C01815=1196.724,348.587,-75.076,-176.172,7.976,148.435
C01816=1196.728,348.340,-75.043,-176.174,7.973,148.435
C01817=1196.731,348.092,-75.011,-176.176,7.970,148.435
C01818=1196.736,347.844,-74.978,-176.177,7.966,148.434
C01819=1196.740,347.596,-74.944,-176.180,7.963,148.434
C01820=1196.745,347.348,-74.912,-176.182,7.960,148.434
C01821=1196.749,347.101,-74.879,-176.184,7.957,148.434
C01822=1196.753,346.853,-74.847,-176.186,7.954,148.433
C01823=1196.757,346.605,-74.814,-176.188,7.951,148.433
C01824=1196.761,346.357,-74.781,-176.190,7.947,148.433
C01825=1196.765,346.109,-74.749,-176.192,7.945,148.433
C01826=1196.769,345.862,-74.716,-176.194,7.941,148.433
C01827=1196.773,345.613,-74.684,-176.196,7.938,148.432
C01828=1196.778,345.366,-74.651,-176.199,7.935,148.432
C01829=1196.782,345.118,-74.619,-176.201,7.931,148.432
C01830=1196.786,344.870,-74.586,-176.202,7.929,148.432
C01831=1196.790,344.622,-74.553,-176.205,7.926,148.431
C01832=1196.794,344.375,-74.521,-176.207,7.922,148.431
C01833=1196.798,344.126,-74.488,-176.209,7.919,148.431
C01834=1196.802,343.879,-74.455,-176.211,7.916,148.431
C01835=1196.807,343.631,-74.424,-176.213,7.913,148.431
C01836=1196.811,343.383,-74.391,-176.216,7.910,148.431
C01837=1196.815,343.135,-74.358,-176.218,7.907,148.430
C01838=1196.819,342.888,-74.326,-176.220,7.904,148.430
C01839=1196.823,342.639,-74.293,-176.222,7.901,148.430
C01840=1196.827,342.391,-74.261,-176.224,7.898,148.430
C01841=1196.831,342.144,-74.228,-176.226,7.894,148.430
C01842=1196.836,341.896,-74.196,-176.228,7.892,148.429
C01843=1196.839,341.648,-74.163,-176.230,7.888,148.429
C01844=1196.844,341.400,-74.131,-176.233,7.885,148.429
C01845=1196.848,341.152,-74.099,-176.235,7.882,148.429
C01846=1196.853,340.874,-74.062,-176.237,7.879,148.429
C01847=1196.858,340.595,-74.026,-176.240,7.875,148.429
C01848=1196.862,340.317,-73.989,-176.242,7.872,148.428
C01849=1196.867,340.038,-73.954,-176.245,7.868,148.428
C01850=1196.871,339.791,-73.921,-176.246,7.865,148.428
C01851=1196.875,339.543,-73.889,-176.249,7.862,148.428
C01852=1196.879,339.295,-73.857,-176.251,7.859,148.428
C01853=1196.883,339.046,-73.824,-176.254,7.856,148.427
C01854=1196.887,338.799,-73.792,-176.255,7.853,148.427
C01855=1196.892,338.551,-73.760,-176.257,7.850,148.427
C01856=1196.896,338.303,-73.728,-176.260,7.847,148.427
C01857=1196.901,338.055,-73.696,-176.262,7.843,148.427
C01858=1196.904,337.807,-73.664,-176.264,7.841,148.427
C01859=1196.908,337.559,-73.632,-176.266,7.838,148.426
C01860=1196.912,337.312,-73.599,-176.269,7.835,148.426
C01861=1196.917,337.064,-73.568,-176.271,7.831,148.426
C01862=1196.921,336.816,-73.535,-176.273,7.829,148.426
C01863=1196.925,336.568,-73.503,-176.275,7.825,148.426
C01864=1196.929,336.320,-73.471,-176.278,7.822,148.426
C01865=1196.933,336.072,-73.439,-176.280,7.819,148.426
C01866=1196.937,335.824,-73.408,-176.282,7.816,148.425
C01867=1196.942,335.576,-73.375,-176.284,7.813,148.425
C01868=1196.946,335.329,-73.344,-176.287,7.810,148.425
C01869=1196.950,335.080,-73.311,-176.289,7.807,148.425
C01870=1196.954,334.832,-73.279,-176.291,7.804,148.425
C01871=1196.958,334.585,-73.248,-176.293,7.801,148.425
C01872=1196.963,334.336,-73.215,-176.295,7.798,148.425
C01873=1196.966,334.088,-73.184,-176.298,7.795,148.424
C01874=1196.971,333.841,-73.152,-176.300,7.792,148.424
C01875=1196.975,333.593,-73.120,-176.302,7.789,148.424
C01876=1196.979,333.345,-73.088,-176.304,7.786,148.424
C01877=1196.983,333.097,-73.056,-176.307,7.783,148.424
C01878=1196.988,332.849,-73.024,-176.309,7.780,148.424
C01879=1196.991,332.601,-72.992,-176.311,7.777,148.424
C01880=1196.996,332.354,-72.961,-176.314,7.774,148.424
C01881=1196.999,332.106,-72.929,-176.316,7.771,148.423
C01882=1197.004,331.858,-72.897,-176.318,7.768,148.423
C01883=1197.008,331.609,-72.865,-176.320,7.765,148.423
C01884=1197.012,331.361,-72.834,-176.322,7.762,148.423
C01885=1197.017,331.114,-72.802,-176.325,7.759,148.423
C01886=1197.021,330.866,-72.770,-176.327,7.755,148.423
C01887=1197.025,330.618,-72.738,-176.329,7.753,148.423
C01888=1197.029,330.370,-72.706,-176.332,7.750,148.423
C01889=1197.033,330.121,-72.675,-176.334,7.747,148.422
C01890=1197.038,329.874,-72.643,-176.337,7.744,148.422
C01891=1197.042,329.626,-72.611,-176.339,7.740,148.422
C01892=1197.046,329.378,-72.580,-176.341,7.738,148.422
C01893=1197.050,329.130,-72.549,-176.343,7.735,148.422
C01894=1197.054,328.882,-72.517,-176.346,7.732,148.422
C01895=1197.059,328.634,-72.485,-176.348,7.728,148.422
C01896=1197.062,328.386,-72.453,-176.350,7.726,148.422
C01897=1197.067,328.138,-72.422,-176.352,7.723,148.422
C01898=1197.071,327.890,-72.390,-176.355,7.720,148.421
C01899=1197.075,327.643,-72.359,-176.357,7.716,148.421
C01900=1197.079,327.394,-72.328,-176.359,7.714,148.421
C01901=1197.084,327.146,-72.296,-176.362,7.711,148.421
C01902=1197.088,326.898,-72.265,-176.364,7.708,148.421
C01903=1197.092,326.650,-72.233,-176.367,7.705,148.421
C01904=1197.096,326.402,-72.201,-176.368,7.702,148.421
C01905=1197.101,326.154,-72.170,-176.371,7.699,148.421
C01906=1197.105,325.906,-72.139,-176.373,7.696,148.421
C01907=1197.109,325.658,-72.108,-176.376,7.693,148.421
C01908=1197.113,325.410,-72.076,-176.378,7.691,148.421
C01909=1197.117,325.162,-72.045,-176.380,7.687,148.420
C01910=1197.121,324.914,-72.013,-176.383,7.684,148.420
C01911=1197.125,324.667,-71.982,-176.385,7.681,148.420
C01912=1197.129,324.418,-71.951,-176.387,7.679,148.420
C01913=1197.134,324.171,-71.919,-176.390,7.675,148.420
C01914=1197.138,323.922,-71.888,-176.392,7.672,148.420
C01915=1197.142,323.674,-71.857,-176.394,7.669,148.420
C01916=1197.146,323.426,-71.826,-176.397,7.667,148.420
C01917=1197.151,323.178,-71.795,-176.399,7.664,148.420
C01918=1197.154,322.930,-71.763,-176.402,7.660,148.420
C01919=1197.159,322.682,-71.732,-176.404,7.657,148.420
C01920=1197.163,322.434,-71.700,-176.406,7.655,148.420
C01921=1197.167,322.186,-71.670,-176.409,7.652,148.420
C01922=1197.171,321.938,-71.638,-176.411,7.649,148.420
C01923=1197.176,321.690,-71.607,-176.414,7.646,148.419
C01924=1197.180,321.443,-71.576,-176.416,7.643,148.419
C01925=1197.184,321.194,-71.545,-176.418,7.640,148.419
C01926=1197.189,320.947,-71.514,-176.421,7.637,148.419
C01927=1197.193,320.698,-71.482,-176.423,7.634,148.419
C01928=1197.197,320.450,-71.452,-176.425,7.631,148.419
C01929=1197.202,320.203,-71.420,-176.428,7.628,148.419
C01930=1197.205,319.954,-71.390,-176.430,7.625,148.419
C01931=1197.209,319.706,-71.359,-176.432,7.623,148.419
C01932=1197.213,319.458,-71.328,-176.435,7.620,148.419
C01933=1197.218,319.210,-71.296,-176.437,7.617,148.419
C01934=1197.222,318.962,-71.266,-176.440,7.614,148.419
C01935=1197.226,318.714,-71.234,-176.442,7.611,148.419
C01936=1197.231,318.466,-71.204,-176.444,7.608,148.419
C01937=1197.234,318.217,-71.173,-176.447,7.605,148.419
C01938=1197.239,317.970,-71.142,-176.449,7.602,148.419
C01939=1197.243,317.722,-71.111,-176.451,7.600,148.418
C01940=1197.247,317.473,-71.080,-176.454,7.596,148.418
C01941=1197.252,317.225,-71.049,-176.456,7.593,148.418
C01942=1197.256,316.977,-71.018,-176.459,7.590,148.418
C01943=1197.260,316.729,-70.988,-176.461,7.588,148.418
C01944=1197.264,316.481,-70.957,-176.464,7.585,148.418
C01945=1197.269,316.234,-70.925,-176.466,7.582,148.418
C01946=1197.273,315.985,-70.894,-176.468,7.579,148.418
C01947=1197.277,315.738,-70.864,-176.471,7.576,148.418
C01948=1197.281,315.490,-70.833,-176.473,7.573,148.418
C01949=1197.286,315.242,-70.803,-176.476,7.570,148.418
C01950=1197.290,314.964,-70.769,-176.478,7.567,148.418
C01951=1197.295,314.689,-70.734,-176.481,7.564,148.418
C01952=1197.299,314.412,-70.700,-176.484,7.561,148.418
C01953=1197.304,314.136,-70.666,-176.486,7.558,148.418
C01954=1197.309,313.888,-70.635,-176.489,7.555,148.418
C01955=1197.313,313.639,-70.604,-176.491,7.552,148.418
C01956=1197.317,313.392,-70.574,-176.493,7.549,148.418
C01957=1197.321,313.144,-70.543,-176.496,7.546,148.418
C01958=1197.326,312.896,-70.513,-176.499,7.543,148.418
C01959=1197.329,312.647,-70.482,-176.501,7.540,148.418
C01960=1197.334,312.399,-70.451,-176.503,7.538,148.418
C01961=1197.338,312.151,-70.421,-176.506,7.535,148.418
C01962=1197.343,311.903,-70.391,-176.508,7.532,148.418
C01963=1197.347,311.654,-70.360,-176.511,7.530,148.418
C01964=1197.351,311.407,-70.330,-176.513,7.526,148.418
C01965=1197.355,311.159,-70.299,-176.516,7.523,148.418
C01966=1197.360,310.911,-70.268,-176.518,7.520,148.418
C01967=1197.364,310.663,-70.238,-176.520,7.518,148.418
C01968=1197.368,310.414,-70.208,-176.523,7.515,148.417
C01969=1197.372,310.166,-70.178,-176.525,7.512,148.417
C01970=1197.376,309.918,-70.147,-176.527,7.510,148.417
C01971=1197.381,309.670,-70.116,-176.530,7.507,148.418
C01972=1197.385,309.422,-70.087,-176.533,7.504,148.418
C01973=1197.389,309.173,-70.055,-176.536,7.500,148.418
C01974=1197.393,308.926,-70.025,-176.537,7.498,148.417
C01975=1197.398,308.678,-69.994,-176.540,7.495,148.417
C01976=1197.402,308.430,-69.965,-176.543,7.492,148.417
C01977=1197.407,308.182,-69.934,-176.545,7.490,148.417
C01978=1197.410,307.934,-69.904,-176.547,7.487,148.417
C01979=1197.415,307.685,-69.874,-176.550,7.484,148.417
C01980=1197.419,307.437,-69.844,-176.552,7.481,148.417
C01981=1197.423,307.189,-69.813,-176.555,7.478,148.417
C01982=1197.427,306.941,-69.783,-176.557,7.475,148.417
C01983=1197.432,306.693,-69.753,-176.560,7.472,148.417
C01984=1197.436,306.445,-69.723,-176.562,7.470,148.417
C01985=1197.441,306.197,-69.692,-176.565,7.467,148.417
C01986=1197.445,305.948,-69.663,-176.567,7.464,148.417
C01987=1197.449,305.700,-69.632,-176.570,7.462,148.418
C01988=1197.453,305.452,-69.602,-176.572,7.458,148.417
C01989=1197.457,305.204,-69.572,-176.574,7.455,148.417
C01990=1197.462,304.956,-69.541,-176.577,7.453,148.417
C01991=1197.466,304.708,-69.512,-176.579,7.450,148.417
C01992=1197.470,304.460,-69.481,-176.582,7.447,148.417
C01993=1197.475,304.211,-69.452,-176.585,7.444,148.417
C01994=1197.479,303.964,-69.422,-176.587,7.442,148.417
C01995=1197.483,303.715,-69.391,-176.590,7.439,148.418
C01996=1197.488,303.467,-69.362,-176.592,7.436,148.418
C01997=1197.492,303.219,-69.331,-176.594,7.434,148.418
C01998=1197.496,302.971,-69.302,-176.597,7.430,148.417
C01999=1197.500,302.723,-69.272,-176.599,7.427,148.417
C02000=1197.505,302.474,-69.241,-176.601,7.425,148.417
C02001=1197.509,302.225,-69.212,-176.604,7.422,148.417
C02002=1197.513,301.978,-69.182,-176.607,7.419,148.417
C02003=1197.518,301.729,-69.152,-176.609,7.417,148.418
C02004=1197.522,301.481,-69.122,-176.612,7.414,148.418
C02005=1197.526,301.233,-69.092,-176.614,7.411,148.418
C02006=1197.530,300.985,-69.062,-176.617,7.409,148.418
C02007=1197.535,300.736,-69.032,-176.619,7.406,148.418
C02008=1197.539,300.489,-69.002,-176.622,7.403,148.418
C02009=1197.543,300.241,-68.973,-176.624,7.401,148.418
C02010=1197.547,299.992,-68.943,-176.627,7.398,148.418
C02011=1197.552,299.744,-68.913,-176.629,7.395,148.418
C02012=1197.556,299.496,-68.883,-176.632,7.392,148.418
C02013=1197.560,299.248,-68.854,-176.634,7.389,148.418
C02014=1197.564,298.999,-68.824,-176.637,7.386,148.418
C02015=1197.569,298.751,-68.794,-176.639,7.384,148.418
C02016=1197.573,298.503,-68.764,-176.642,7.381,148.418
C02017=1197.577,298.255,-68.735,-176.645,7.378,148.418
C02018=1197.581,298.007,-68.705,-176.646,7.376,148.418
C02019=1197.586,297.758,-68.676,-176.649,7.373,148.418
C02020=1197.590,297.510,-68.646,-176.652,7.370,148.418
C02021=1197.595,297.262,-68.617,-176.654,7.367,148.418
C02022=1197.599,297.014,-68.587,-176.656,7.364,148.418
C02023=1197.603,296.766,-68.557,-176.659,7.361,148.418
C02024=1197.607,296.518,-68.527,-176.661,7.359,148.418
C02025=1197.612,296.270,-68.498,-176.664,7.356,148.418
C02026=1197.616,296.022,-68.469,-176.667,7.353,148.418
C02027=1197.620,295.773,-68.439,-176.669,7.351,148.418
C02028=1197.624,295.525,-68.410,-176.672,7.348,148.418
C02029=1197.629,295.276,-68.380,-176.674,7.346,148.418
C02030=1197.633,295.028,-68.350,-176.677,7.343,148.418
C02031=1197.637,294.780,-68.321,-176.680,7.340,148.419
C02032=1197.642,294.532,-68.291,-176.682,7.338,148.419
C02033=1197.646,294.283,-68.262,-176.684,7.335,148.419
C02034=1197.651,294.036,-68.233,-176.687,7.332,148.419
C02035=1197.655,293.788,-68.203,-176.689,7.330,148.419
C02036=1197.659,293.539,-68.174,-176.692,7.327,148.419
C02037=1197.663,293.291,-68.144,-176.695,7.324,148.419
C02038=1197.667,293.043,-68.115,-176.697,7.322,148.419
C02039=1197.672,292.794,-68.086,-176.699,7.318,148.419
C02040=1197.676,292.546,-68.057,-176.702,7.316,148.419
C02041=1197.680,292.297,-68.027,-176.704,7.313,148.419
C02042=1197.685,292.050,-67.998,-176.707,7.310,148.419
C02043=1197.689,291.802,-67.969,-176.709,7.308,148.419
C02044=1197.693,291.553,-67.939,-176.712,7.305,148.419
C02045=1197.698,291.305,-67.910,-176.715,7.302,148.419
C02046=1197.702,291.056,-67.881,-176.717,7.300,148.419
C02047=1197.706,290.808,-67.852,-176.719,7.297,148.419
C02048=1197.711,290.560,-67.822,-176.722,7.295,148.419
C02049=1197.715,290.312,-67.793,-176.725,7.292,148.419
C02050=1197.719,290.064,-67.764,-176.727,7.289,148.419
C02051=1197.724,289.815,-67.735,-176.730,7.287,148.420
C02052=1197.727,289.567,-67.706,-176.732,7.284,148.420
C02053=1197.732,289.319,-67.677,-176.734,7.282,148.420
C02054=1197.737,289.044,-67.644,-176.737,7.279,148.420
C02055=1197.742,288.770,-67.613,-176.740,7.276,148.420
C02056=1197.746,288.496,-67.580,-176.743,7.273,148.420
C02057=1197.751,288.221,-67.549,-176.746,7.270,148.420
C02058=1197.755,287.973,-67.519,-176.748,7.267,148.420
C02059=1197.760,287.724,-67.490,-176.751,7.264,148.420
C02060=1197.764,287.476,-67.461,-176.753,7.262,148.420
C02061=1197.769,287.228,-67.432,-176.756,7.259,148.420
C02062=1197.773,286.980,-67.403,-176.758,7.256,148.420
C02063=1197.777,286.731,-67.374,-176.761,7.253,148.420
C02064=1197.781,286.483,-67.346,-176.764,7.251,148.420
C02065=1197.786,286.235,-67.317,-176.766,7.249,148.421
C02066=1197.790,285.987,-67.287,-176.769,7.246,148.421
C02067=1197.795,285.738,-67.258,-176.771,7.243,148.421
C02068=1197.799,285.490,-67.229,-176.774,7.240,148.421
C02069=1197.803,285.242,-67.201,-176.776,7.237,148.421
C02070=1197.807,284.994,-67.172,-176.778,7.235,148.421
C02071=1197.812,284.745,-67.143,-176.782,7.233,148.421
C02072=1197.817,284.497,-67.114,-176.784,7.230,148.421
C02073=1197.820,284.249,-67.086,-176.787,7.227,148.421
C02074=1197.825,284.000,-67.056,-176.789,7.225,148.421
C02075=1197.830,283.752,-67.028,-176.791,7.222,148.421
C02076=1197.833,283.504,-66.999,-176.794,7.219,148.421
C02077=1197.838,283.255,-66.970,-176.796,7.217,148.421
C02078=1197.843,283.007,-66.942,-176.799,7.214,148.422
C02079=1197.847,282.759,-66.912,-176.802,7.212,148.422
C02080=1197.851,282.510,-66.884,-176.804,7.209,148.422
C02081=1197.855,282.263,-66.855,-176.806,7.207,148.422
C02082=1197.860,282.014,-66.826,-176.809,7.204,148.422
C02083=1197.864,281.765,-66.798,-176.812,7.201,148.422
C02084=1197.868,281.518,-66.769,-176.814,7.199,148.422
C02085=1197.873,281.269,-66.740,-176.817,7.196,148.422
C02086=1197.877,281.020,-66.712,-176.819,7.194,148.422
C02087=1197.881,280.773,-66.683,-176.822,7.191,148.422
C02088=1197.885,280.524,-66.655,-176.824,7.189,148.422
C02089=1197.890,280.275,-66.626,-176.827,7.186,148.423
C02090=1197.895,280.027,-66.598,-176.830,7.183,148.423
C02091=1197.898,279.779,-66.569,-176.832,7.181,148.423
C02092=1197.903,279.531,-66.541,-176.835,7.178,148.423
C02093=1197.907,279.282,-66.513,-176.837,7.176,148.423
C02094=1197.911,279.033,-66.484,-176.840,7.173,148.423
C02095=1197.916,278.786,-66.456,-176.842,7.171,148.423
C02096=1197.920,278.537,-66.427,-176.845,7.168,148.423
C02097=1197.925,278.289,-66.398,-176.847,7.166,148.423
C02098=1197.929,278.040,-66.370,-176.850,7.163,148.423
C02099=1197.934,277.792,-66.342,-176.852,7.161,148.424
C02100=1197.938,277.544,-66.314,-176.855,7.158,148.424
C02101=1197.942,277.295,-66.285,-176.858,7.155,148.424
C02102=1197.946,277.048,-66.256,-176.860,7.152,148.424
C02103=1197.951,276.799,-66.228,-176.863,7.149,148.424
C02104=1197.955,276.551,-66.200,-176.865,7.148,148.424
C02105=1197.960,276.302,-66.171,-176.868,7.145,148.424
C02106=1197.964,276.054,-66.143,-176.870,7.142,148.424
C02107=1197.968,275.805,-66.115,-176.873,7.139,148.424
C02108=1197.973,275.557,-66.087,-176.876,7.138,148.424
C02109=1197.976,275.309,-66.059,-176.878,7.135,148.424
C02110=1197.982,275.061,-66.030,-176.880,7.132,148.425
C02111=1197.985,274.812,-66.002,-176.883,7.129,148.425
C02112=1197.990,274.564,-65.974,-176.886,7.127,148.425
C02113=1197.994,274.315,-65.946,-176.888,7.124,148.425
C02114=1197.999,274.067,-65.917,-176.891,7.122,148.425
C02115=1198.003,273.818,-65.889,-176.893,7.119,148.425
C02116=1198.007,273.571,-65.861,-176.896,7.117,148.425
C02117=1198.012,273.322,-65.833,-176.899,7.114,148.425
C02118=1198.016,273.074,-65.805,-176.901,7.112,148.425
C02119=1198.020,272.825,-65.777,-176.903,7.109,148.425
C02120=1198.025,272.577,-65.748,-176.906,7.107,148.426
C02121=1198.029,272.328,-65.721,-176.909,7.104,148.426
C02122=1198.034,272.080,-65.693,-176.911,7.102,148.426
C02123=1198.038,271.831,-65.664,-176.914,7.100,148.426
C02124=1198.042,271.583,-65.637,-176.916,7.097,148.426
C02125=1198.047,271.334,-65.608,-176.919,7.094,148.426
C02126=1198.051,271.086,-65.580,-176.921,7.092,148.426
C02127=1198.055,270.839,-65.552,-176.924,7.089,148.427
C02128=1198.059,270.589,-65.525,-176.926,7.087,148.427
C02129=1198.065,270.341,-65.497,-176.929,7.084,148.427
C02130=1198.068,270.093,-65.468,-176.931,7.082,148.427
C02131=1198.073,269.845,-65.441,-176.934,7.079,148.427
C02132=1198.077,269.595,-65.413,-176.937,7.077,148.427
C02133=1198.082,269.347,-65.385,-176.939,7.074,148.427
C02134=1198.086,269.099,-65.357,-176.942,7.072,148.427
C02135=1198.090,268.851,-65.329,-176.945,7.069,148.428
C02136=1198.095,268.602,-65.301,-176.947,7.067,148.428
C02137=1198.099,268.353,-65.273,-176.950,7.065,148.428
C02138=1198.103,268.106,-65.245,-176.952,7.062,148.428
C02139=1198.108,267.857,-65.218,-176.955,7.059,148.428
C02140=1198.112,267.609,-65.190,-176.957,7.058,148.428
C02141=1198.117,267.360,-65.162,-176.960,7.054,148.428
C02142=1198.122,267.112,-65.135,-176.962,7.052,148.428
C02143=1198.125,266.863,-65.107,-176.965,7.050,148.429
C02144=1198.130,266.615,-65.079,-176.968,7.047,148.429
C02145=1198.134,266.367,-65.052,-176.970,7.044,148.429
C02146=1198.138,266.118,-65.024,-176.973,7.043,148.429
C02147=1198.143,265.870,-64.996,-176.975,7.040,148.429
C02148=1198.148,265.622,-64.968,-176.978,7.037,148.429
C02149=1198.152,265.372,-64.941,-176.980,7.036,148.430
C02150=1198.156,265.125,-64.913,-176.983,7.033,148.430
C02151=1198.161,264.876,-64.886,-176.985,7.030,148.430
C02152=1198.165,264.628,-64.858,-176.988,7.028,148.430
C02153=1198.169,264.379,-64.831,-176.991,7.026,148.430
C02154=1198.174,264.131,-64.803,-176.993,7.023,148.430
C02155=1198.178,263.882,-64.775,-176.996,7.021,148.430
C02156=1198.183,263.634,-64.747,-176.998,7.019,148.430
C02157=1198.187,263.385,-64.720,-177.001,7.016,148.430
C02158=1198.191,263.112,-64.690,-177.004,7.013,148.431
C02159=1198.197,262.840,-64.660,-177.006,7.011,148.431
C02160=1198.202,262.567,-64.629,-177.009,7.008,148.431
C02161=1198.206,262.294,-64.599,-177.012,7.005,148.431
C02162=1198.210,262.045,-64.572,-177.015,7.003,148.431
C02163=1198.215,261.798,-64.544,-177.017,7.000,148.431
C02164=1198.219,261.549,-64.517,-177.020,6.998,148.432
C02165=1198.224,261.300,-64.490,-177.023,6.995,148.432
C02166=1198.228,261.052,-64.462,-177.025,6.993,148.432
C02167=1198.233,260.804,-64.435,-177.028,6.990,148.432
C02168=1198.237,260.555,-64.408,-177.030,6.988,148.432
C02169=1198.241,260.306,-64.380,-177.032,6.986,148.432
C02170=1198.246,260.058,-64.353,-177.036,6.983,148.433
C02171=1198.250,259.809,-64.326,-177.038,6.981,148.433
C02172=1198.255,259.561,-64.299,-177.040,6.978,148.433
C02173=1198.259,259.313,-64.271,-177.043,6.976,148.433
C02174=1198.263,259.064,-64.243,-177.046,6.973,148.433
C02175=1198.268,258.815,-64.216,-177.048,6.972,148.433
C02176=1198.273,258.567,-64.189,-177.051,6.969,148.434
C02177=1198.277,258.319,-64.162,-177.053,6.966,148.434
C02178=1198.282,258.071,-64.135,-177.056,6.964,148.434
C02179=1198.286,257.821,-64.107,-177.059,6.961,148.434
C02180=1198.290,257.573,-64.081,-177.061,6.960,148.434
C02181=1198.294,257.325,-64.054,-177.063,6.957,148.434
C02182=1198.299,257.076,-64.027,-177.067,6.955,148.435
C02183=1198.304,256.828,-63.999,-177.069,6.953,148.435
C02184=1198.308,256.580,-63.972,-177.071,6.950,148.435
C02185=1198.312,256.331,-63.944,-177.074,6.948,148.435
C02186=1198.317,256.082,-63.917,-177.076,6.946,148.435
C02187=1198.321,255.834,-63.891,-177.079,6.943,148.435
C02188=1198.325,255.585,-63.864,-177.082,6.941,148.435
C02189=1198.330,255.337,-63.837,-177.084,6.939,148.436
C02190=1198.335,255.088,-63.810,-177.087,6.936,148.436
C02191=1198.339,254.840,-63.782,-177.089,6.934,148.436
C02192=1198.343,254.592,-63.756,-177.092,6.931,148.436
C02193=1198.347,254.343,-63.729,-177.094,6.929,148.436
C02194=1198.352,254.094,-63.702,-177.097,6.927,148.437
C02195=1198.357,253.846,-63.674,-177.100,6.924,148.437
C02196=1198.361,253.597,-63.647,-177.102,6.922,148.437
C02197=1198.365,253.349,-63.621,-177.104,6.920,148.437
C02198=1198.370,253.100,-63.594,-177.108,6.917,148.437
C02199=1198.374,252.852,-63.567,-177.110,6.915,148.437
C02200=1198.378,252.604,-63.540,-177.113,6.912,148.437
C02201=1198.383,252.355,-63.513,-177.115,6.910,148.438
C02202=1198.388,252.107,-63.486,-177.117,6.908,148.438
C02203=1198.392,251.858,-63.459,-177.121,6.905,148.438
C02204=1198.396,251.609,-63.433,-177.123,6.903,148.438
C02205=1198.401,251.360,-63.406,-177.125,6.901,148.439
C02206=1198.405,251.112,-63.379,-177.128,6.898,148.439
C02207=1198.409,250.864,-63.352,-177.131,6.897,148.439
C02208=1198.414,250.615,-63.325,-177.133,6.894,148.439
C02209=1198.418,250.367,-63.298,-177.136,6.892,148.439
C02210=1198.423,250.118,-63.273,-177.138,6.890,148.439
C02211=1198.427,249.869,-63.246,-177.141,6.888,148.440
C02212=1198.432,249.621,-63.218,-177.143,6.885,148.440
C02213=1198.436,249.373,-63.192,-177.146,6.883,148.440
C02214=1198.441,249.124,-63.165,-177.149,6.880,148.440
C02215=1198.445,248.875,-63.139,-177.151,6.878,148.440
C02216=1198.449,248.627,-63.112,-177.154,6.876,148.440
C02217=1198.454,248.378,-63.085,-177.157,6.873,148.441
C02218=1198.458,248.130,-63.059,-177.159,6.871,148.441
C02219=1198.463,247.881,-63.032,-177.162,6.869,148.441
C02220=1198.467,247.633,-63.006,-177.164,6.866,148.441
C02221=1198.472,247.384,-62.979,-177.167,6.864,148.442
C02222=1198.476,247.136,-62.953,-177.169,6.862,148.442
C02223=1198.480,246.887,-62.926,-177.172,6.860,148.442
C02224=1198.485,246.639,-62.899,-177.174,6.857,148.442
C02225=1198.489,246.390,-62.873,-177.177,6.856,148.442
C02226=1198.494,246.141,-62.846,-177.179,6.853,148.442
C02227=1198.498,245.892,-62.820,-177.182,6.851,148.443
C02228=1198.503,245.644,-62.793,-177.185,6.849,148.443
C02229=1198.507,245.396,-62.767,-177.187,6.847,148.443
C02230=1198.512,245.147,-62.741,-177.190,6.844,148.443
C02231=1198.516,244.899,-62.714,-177.193,6.842,148.443
C02232=1198.521,244.650,-62.688,-177.195,6.840,148.444
C02233=1198.525,244.402,-62.661,-177.198,6.837,148.444
C02234=1198.530,244.153,-62.635,-177.200,6.835,148.444
C02235=1198.534,243.905,-62.609,-177.203,6.833,148.444
C02236=1198.538,243.656,-62.583,-177.205,6.830,148.444
C02237=1198.543,243.407,-62.556,-177.208,6.828,148.445
C02238=1198.547,243.158,-62.530,-177.210,6.826,148.445
C02239=1198.552,242.910,-62.503,-177.213,6.824,148.445
C02240=1198.556,242.661,-62.477,-177.216,6.822,148.445
C02241=1198.561,242.413,-62.450,-177.218,6.819,148.445
C02242=1198.565,242.165,-62.425,-177.221,6.818,148.446
C02243=1198.569,241.916,-62.398,-177.224,6.815,148.446
C02244=1198.574,241.667,-62.372,-177.226,6.813,148.446
C02245=1198.579,241.418,-62.346,-177.228,6.810,148.446
C02246=1198.583,241.170,-62.320,-177.232,6.808,148.447
C02247=1198.587,240.921,-62.293,-177.234,6.806,148.447
C02248=1198.592,240.672,-62.268,-177.236,6.804,148.447
C02249=1198.597,240.425,-62.241,-177.239,6.802,148.447
C02250=1198.601,240.176,-62.215,-177.242,6.799,148.447
C02251=1198.605,239.927,-62.190,-177.244,6.797,148.448
C02252=1198.610,239.678,-62.162,-177.246,6.795,148.448
C02253=1198.614,239.430,-62.137,-177.249,6.793,148.448
C02254=1198.619,239.181,-62.111,-177.252,6.790,148.448
C02255=1198.623,238.933,-62.085,-177.254,6.788,148.448
C02256=1198.628,238.684,-62.059,-177.257,6.786,148.449
C02257=1198.632,238.435,-62.033,-177.260,6.783,148.449
C02258=1198.636,238.187,-62.007,-177.262,6.782,148.449
C02259=1198.641,237.938,-61.980,-177.265,6.779,148.449
C02260=1198.646,237.690,-61.955,-177.267,6.778,148.450
C02261=1198.650,237.441,-61.929,-177.270,6.775,148.450
C02262=1198.655,237.169,-61.901,-177.273,6.773,148.450
C02263=1198.659,236.898,-61.872,-177.276,6.770,148.450
C02264=1198.665,236.627,-61.844,-177.278,6.768,148.451
C02265=1198.670,236.355,-61.815,-177.282,6.766,148.451
C02266=1198.674,236.106,-61.789,-177.284,6.763,148.451
C02267=1198.678,235.858,-61.763,-177.286,6.762,148.451
C02268=1198.683,235.610,-61.738,-177.289,6.759,148.451
C02269=1198.688,235.360,-61.712,-177.292,6.757,148.452
C02270=1198.692,235.112,-61.686,-177.294,6.755,148.452
C02271=1198.696,234.863,-61.660,-177.297,6.753,148.452
C02272=1198.701,234.615,-61.635,-177.300,6.750,148.452
C02273=1198.705,234.367,-61.608,-177.302,6.748,148.453
C02274=1198.709,234.118,-61.583,-177.305,6.746,148.453
C02275=1198.715,233.869,-61.557,-177.307,6.744,148.453
C02276=1198.719,233.620,-61.531,-177.310,6.741,148.453
C02277=1198.723,233.372,-61.505,-177.313,6.739,148.453
C02278=1198.728,233.123,-61.479,-177.315,6.738,148.454
C02279=1198.732,232.875,-61.454,-177.317,6.735,148.454
C02280=1198.737,232.626,-61.428,-177.320,6.734,148.454
C02281=1198.741,232.377,-61.403,-177.323,6.731,148.455
C02282=1198.746,232.129,-61.377,-177.325,6.729,148.455
C02283=1198.750,231.880,-61.351,-177.328,6.727,148.455
C02284=1198.755,231.631,-61.325,-177.331,6.725,148.455
C02285=1198.760,231.382,-61.300,-177.333,6.722,148.455
C02286=1198.764,231.134,-61.275,-177.336,6.720,148.456
C02287=1198.768,230.885,-61.249,-177.339,6.718,148.456
C02288=1198.773,230.637,-61.223,-177.341,6.716,148.456
C02289=1198.777,230.388,-61.198,-177.343,6.715,148.456
C02290=1198.782,230.139,-61.172,-177.347,6.712,148.457
C02291=1198.787,229.891,-61.147,-177.349,6.710,148.457
C02292=1198.791,229.642,-61.121,-177.351,6.708,148.457
C02293=1198.795,229.393,-61.096,-177.354,6.706,148.457
C02294=1198.800,229.145,-61.070,-177.357,6.703,148.458
C02295=1198.804,228.896,-61.045,-177.359,6.701,148.458
C02296=1198.809,228.647,-61.019,-177.362,6.699,148.458
C02297=1198.813,228.399,-60.994,-177.364,6.697,148.458
C02298=1198.818,228.150,-60.969,-177.367,6.695,148.459
C02299=1198.823,227.901,-60.943,-177.370,6.693,148.459
C02300=1198.827,227.653,-60.917,-177.372,6.691,148.459
C02301=1198.831,227.404,-60.892,-177.375,6.689,148.459
C02302=1198.836,227.155,-60.867,-177.378,6.687,148.460
C02303=1198.840,226.907,-60.842,-177.380,6.685,148.460
C02304=1198.845,226.658,-60.816,-177.383,6.682,148.460
C02305=1198.849,226.410,-60.791,-177.386,6.680,148.460
C02306=1198.853,226.160,-60.766,-177.388,6.678,148.460
C02307=1198.858,225.912,-60.740,-177.390,6.676,148.461
C02308=1198.862,225.663,-60.714,-177.393,6.674,148.461
C02309=1198.868,225.415,-60.690,-177.396,6.672,148.461
C02310=1198.872,225.166,-60.664,-177.398,6.670,148.462
C02311=1198.877,224.917,-60.639,-177.401,6.668,148.462
C02312=1198.880,224.669,-60.614,-177.404,6.666,148.462
C02313=1198.885,224.420,-60.589,-177.406,6.664,148.462
C02314=1198.890,224.171,-60.564,-177.408,6.662,148.463
C02315=1198.894,223.922,-60.538,-177.412,6.659,148.463
C02316=1198.899,223.674,-60.513,-177.414,6.657,148.463
C02317=1198.903,223.425,-60.488,-177.416,6.655,148.463
C02318=1198.907,223.177,-60.463,-177.419,6.653,148.464
C02319=1198.912,222.928,-60.438,-177.422,6.652,148.464
C02320=1198.917,222.679,-60.412,-177.424,6.649,148.464
C02321=1198.921,222.430,-60.387,-177.427,6.647,148.464
C02322=1198.926,222.182,-60.362,-177.430,6.645,148.465
C02323=1198.930,221.933,-60.338,-177.432,6.643,148.465
C02324=1198.935,221.685,-60.312,-177.435,6.641,148.465
C02325=1198.939,221.435,-60.287,-177.437,6.639,148.466
C02326=1198.944,221.187,-60.263,-177.440,6.637,148.466
C02327=1198.948,220.938,-60.237,-177.443,6.635,148.466
C02328=1198.953,220.689,-60.213,-177.445,6.633,148.466
C02329=1198.957,220.440,-60.187,-177.448,6.631,148.467
C02330=1198.962,220.192,-60.162,-177.451,6.629,148.467
C02331=1198.966,219.944,-60.137,-177.453,6.627,148.467
C02332=1198.971,219.695,-60.112,-177.456,6.624,148.467
C02333=1198.976,219.446,-60.088,-177.459,6.622,148.468
C02334=1198.980,219.197,-60.063,-177.461,6.620,148.468
C02335=1198.985,218.949,-60.038,-177.464,6.619,148.468
C02336=1198.989,218.699,-60.013,-177.466,6.616,148.468
C02337=1198.993,218.451,-59.988,-177.469,6.615,148.469
C02338=1198.998,218.202,-59.963,-177.471,6.613,148.469
C02339=1199.003,217.953,-59.938,-177.474,6.610,148.469
C02340=1199.007,217.705,-59.914,-177.477,6.608,148.470
C02341=1199.012,217.456,-59.889,-177.479,6.606,148.470
C02342=1199.017,217.207,-59.864,-177.482,6.604,148.470
C02343=1199.021,216.958,-59.839,-177.485,6.602,148.471
C02344=1199.025,216.710,-59.814,-177.487,6.601,148.471
C02345=1199.031,216.461,-59.789,-177.490,6.598,148.471
C02346=1199.034,216.212,-59.765,-177.493,6.596,148.471
C02347=1199.039,215.964,-59.740,-177.495,6.594,148.472
C02348=1199.043,215.715,-59.715,-177.498,6.592,148.472
C02349=1199.048,215.466,-59.690,-177.501,6.590,148.472
C02350=1199.052,215.218,-59.666,-177.503,6.588,148.472
C02351=1199.057,214.968,-59.641,-177.505,6.586,148.473
C02352=1199.062,214.720,-59.617,-177.509,6.584,148.473
C02353=1199.067,214.471,-59.593,-177.511,6.582,148.473
C02354=1199.071,214.223,-59.567,-177.514,6.580,148.474
C02355=1199.075,213.974,-59.543,-177.516,6.578,148.474
C02356=1199.080,213.725,-59.518,-177.519,6.576,148.474
C02357=1199.084,213.476,-59.494,-177.521,6.574,148.474
C02358=1199.089,213.228,-59.469,-177.524,6.572,148.475
C02359=1199.093,212.978,-59.445,-177.527,6.571,148.475
C02360=1199.098,212.730,-59.420,-177.529,6.568,148.475
C02361=1199.103,212.481,-59.396,-177.532,6.566,148.476
C02362=1199.108,212.233,-59.371,-177.535,6.564,148.476
C02363=1199.111,211.983,-59.347,-177.537,6.562,148.476
C02364=1199.117,211.735,-59.322,-177.540,6.560,148.477
C02365=1199.121,211.486,-59.298,-177.543,6.559,148.477
C02366=1199.126,211.215,-59.271,-177.546,6.556,148.477
C02367=1199.131,210.945,-59.244,-177.548,6.554,148.478
C02368=1199.136,210.675,-59.217,-177.551,6.552,148.478
C02369=1199.140,210.405,-59.191,-177.554,6.550,148.478
C02370=1199.145,210.155,-59.167,-177.556,6.547,148.478
C02371=1199.149,209.907,-59.143,-177.559,6.546,148.479
C02372=1199.155,209.658,-59.118,-177.562,6.544,148.479
C02373=1199.159,209.410,-59.094,-177.564,6.542,148.479
C02374=1199.163,209.161,-59.070,-177.567,6.540,148.480
C02375=1199.168,208.912,-59.045,-177.570,6.538,148.480
C02376=1199.172,208.663,-59.021,-177.572,6.536,148.480
C02377=1199.177,208.415,-58.996,-177.575,6.534,148.480
C02378=1199.181,208.166,-58.972,-177.578,6.532,148.481
C02379=1199.186,207.917,-58.949,-177.580,6.530,148.481
C02380=1199.191,207.668,-58.924,-177.583,6.528,148.481
C02381=1199.195,207.419,-58.900,-177.586,6.526,148.482
C02382=1199.199,207.170,-58.875,-177.588,6.524,148.482
C02383=1199.204,206.922,-58.851,-177.591,6.522,148.482
C02384=1199.209,206.673,-58.827,-177.593,6.520,148.483
C02385=1199.214,206.424,-58.803,-177.596,6.519,148.483
C02386=1199.219,206.175,-58.779,-177.598,6.517,148.483
C02387=1199.222,205.926,-58.754,-177.601,6.515,148.484
C02388=1199.227,205.678,-58.730,-177.604,6.513,148.484
C02389=1199.232,205.429,-58.707,-177.606,6.511,148.484
C02390=1199.237,205.180,-58.682,-177.609,6.509,148.484
C02391=1199.241,204.932,-58.658,-177.612,6.507,148.485
C02392=1199.246,204.683,-58.635,-177.614,6.505,148.485
C02393=1199.250,204.434,-58.610,-177.617,6.503,148.485
C02394=1199.255,204.185,-58.586,-177.620,6.501,148.486
C02395=1199.259,203.936,-58.561,-177.622,6.499,148.486
C02396=1199.264,203.687,-58.538,-177.625,6.497,148.486
C02397=1199.268,203.439,-58.514,-177.627,6.495,148.487
C02398=1199.274,203.190,-58.490,-177.630,6.493,148.487
C02399=1199.277,202.941,-58.466,-177.633,6.492,148.487
C02400=1199.282,202.692,-58.442,-177.635,6.490,148.488
C02401=1199.286,202.443,-58.418,-177.638,6.488,148.488
C02402=1199.291,202.195,-58.394,-177.640,6.486,148.488
C02403=1199.296,201.946,-58.371,-177.643,6.484,148.489
C02404=1199.301,201.697,-58.346,-177.646,6.483,148.489
C02405=1199.305,201.449,-58.322,-177.648,6.481,148.489
C02406=1199.310,201.199,-58.299,-177.651,6.479,148.489
C02407=1199.314,200.950,-58.274,-177.653,6.477,148.490
C02408=1199.318,200.701,-58.251,-177.656,6.475,148.490
C02409=1199.323,200.453,-58.227,-177.659,6.472,148.490
C02410=1199.327,200.204,-58.203,-177.662,6.471,148.491
C02411=1199.332,199.955,-58.179,-177.664,6.469,148.491
C02412=1199.337,199.706,-58.155,-177.667,6.467,148.491
C02413=1199.342,199.458,-58.131,-177.670,6.465,148.492
C02414=1199.346,199.209,-58.108,-177.672,6.463,148.492
C02415=1199.351,198.960,-58.084,-177.675,6.461,148.492
C02416=1199.355,198.711,-58.061,-177.677,6.459,148.493
C02417=1199.360,198.462,-58.037,-177.680,6.457,148.493
C02418=1199.365,198.214,-58.013,-177.683,6.456,148.493
C02419=1199.369,197.965,-57.990,-177.685,6.454,148.494
C02420=1199.374,197.716,-57.966,-177.688,6.452,148.494
C02421=1199.378,197.467,-57.942,-177.691,6.450,148.494
C02422=1199.382,197.218,-57.919,-177.693,6.448,148.495
C02423=1199.387,196.969,-57.895,-177.696,6.447,148.495
C02424=1199.391,196.720,-57.871,-177.698,6.445,148.495
C02425=1199.396,196.471,-57.848,-177.701,6.443,148.496
C02426=1199.401,196.223,-57.824,-177.704,6.441,148.496
C02427=1199.405,195.974,-57.800,-177.706,6.439,148.496
C02428=1199.410,195.725,-57.777,-177.709,6.438,148.497
C02429=1199.414,195.476,-57.753,-177.711,6.435,148.497
C02430=1199.419,195.227,-57.730,-177.714,6.434,148.497
C02431=1199.424,194.978,-57.706,-177.717,6.432,148.498
C02432=1199.428,194.729,-57.683,-177.719,6.430,148.498
C02433=1199.433,194.481,-57.659,-177.722,6.428,148.498
C02434=1199.438,194.232,-57.635,-177.725,6.426,148.499
C02435=1199.442,193.983,-57.612,-177.727,6.424,148.499
C02436=1199.448,193.734,-57.589,-177.730,6.423,148.499
C02437=1199.452,193.486,-57.565,-177.733,6.421,148.500
C02438=1199.457,193.237,-57.542,-177.735,6.419,148.500
C02439=1199.461,192.988,-57.518,-177.738,6.417,148.500
C02440=1199.465,192.739,-57.496,-177.741,6.415,148.501
C02441=1199.470,192.490,-57.472,-177.743,6.414,148.501
C02442=1199.475,192.241,-57.449,-177.746,6.412,148.501
C02443=1199.479,191.992,-57.425,-177.748,6.410,148.502
C02444=1199.484,191.744,-57.401,-177.751,6.408,148.502
C02445=1199.489,191.495,-57.378,-177.754,6.406,148.502
C02446=1199.493,191.246,-57.355,-177.756,6.405,148.503
C02447=1199.498,190.997,-57.331,-177.759,6.403,148.503
C02448=1199.502,190.748,-57.309,-177.762,6.401,148.504
C02449=1199.507,190.499,-57.285,-177.764,6.399,148.504
C02450=1199.511,190.250,-57.262,-177.767,6.397,148.504
C02451=1199.517,190.001,-57.239,-177.769,6.395,148.504
C02452=1199.521,189.752,-57.215,-177.772,6.393,148.505
C02453=1199.525,189.504,-57.193,-177.775,6.392,148.505
C02454=1199.530,189.255,-57.169,-177.777,6.391,148.505
C02455=1199.535,189.006,-57.146,-177.779,6.389,148.506
C02456=1199.539,188.757,-57.123,-177.782,6.387,148.506
C02457=1199.544,188.508,-57.099,-177.785,6.385,148.506
C02458=1199.548,188.259,-57.076,-177.787,6.383,148.507
C02459=1199.553,188.010,-57.053,-177.790,6.382,148.507
C02460=1199.558,187.761,-57.030,-177.793,6.380,148.508
C02461=1199.563,187.512,-57.007,-177.795,6.378,148.508
C02462=1199.567,187.264,-56.984,-177.798,6.376,148.508
C02463=1199.571,187.015,-56.961,-177.801,6.374,148.509
C02464=1199.576,186.766,-56.937,-177.803,6.372,148.509
C02465=1199.581,186.517,-56.914,-177.806,6.371,148.509
C02466=1199.585,186.269,-56.892,-177.809,6.369,148.510
C02467=1199.590,186.019,-56.869,-177.811,6.367,148.510
C02468=1199.595,185.770,-56.846,-177.814,6.365,148.510
C02469=1199.599,185.521,-56.823,-177.817,6.363,148.511
C02470=1199.604,185.251,-56.798,-177.819,6.362,148.511
C02471=1199.610,184.982,-56.773,-177.822,6.360,148.512
C02472=1199.614,184.712,-56.748,-177.825,6.358,148.512
C02473=1199.620,184.442,-56.723,-177.828,6.357,148.512
C02474=1199.624,184.194,-56.700,-177.830,6.355,148.513
C02475=1199.629,183.945,-56.677,-177.833,6.353,148.513
C02476=1199.634,183.696,-56.654,-177.836,6.351,148.513
C02477=1199.637,183.448,-56.631,-177.838,6.349,148.514
C02478=1199.642,183.198,-56.609,-177.841,6.348,148.514
C02479=1199.646,182.949,-56.586,-177.844,6.346,148.514
C02480=1199.652,182.701,-56.563,-177.846,6.344,148.515
C02481=1199.656,182.452,-56.540,-177.849,6.342,148.515
C02482=1199.661,182.203,-56.518,-177.852,6.340,148.516
C02483=1199.665,181.953,-56.494,-177.854,6.338,148.516
C02484=1199.670,181.705,-56.472,-177.857,6.337,148.516
C02485=1199.675,181.456,-56.449,-177.859,6.336,148.517
C02486=1199.679,181.207,-56.426,-177.862,6.334,148.517
C02487=1199.684,180.958,-56.403,-177.864,6.332,148.517
C02488=1199.689,180.709,-56.381,-177.867,6.330,148.518
C02489=1199.693,180.460,-56.358,-177.870,6.328,148.518
C02490=1199.698,180.211,-56.335,-177.872,6.327,148.518
C02491=1199.703,179.963,-56.313,-177.875,6.325,148.519
C02492=1199.707,179.714,-56.290,-177.878,6.323,148.519
C02493=1199.712,179.464,-56.268,-177.880,6.321,148.520
C02494=1199.716,179.215,-56.244,-177.883,6.319,148.520
C02495=1199.721,178.967,-56.222,-177.886,6.319,148.520
C02496=1199.726,178.718,-56.199,-177.888,6.317,148.521
C02497=1199.730,178.469,-56.176,-177.891,6.315,148.521
C02498=1199.736,178.220,-56.154,-177.894,6.313,148.522
C02499=1199.740,177.971,-56.131,-177.896,6.312,148.522
C02500=1199.744,177.722,-56.109,-177.899,6.310,148.522
C02501=1199.749,177.474,-56.086,-177.902,6.308,148.523
C02502=1199.753,177.224,-56.064,-177.904,6.306,148.523
C02503=1199.758,176.975,-56.041,-177.907,6.304,148.523
C02504=1199.763,176.727,-56.019,-177.909,6.303,148.524
C02505=1199.768,176.477,-55.997,-177.912,6.302,148.524
C02506=1199.772,176.228,-55.974,-177.914,6.300,148.524
C02507=1199.777,175.980,-55.952,-177.917,6.298,148.525
C02508=1199.781,175.731,-55.929,-177.920,6.296,148.525
C02509=1199.786,175.481,-55.907,-177.922,6.294,148.526
C02510=1199.791,175.233,-55.884,-177.925,6.293,148.526
C02511=1199.795,174.983,-55.862,-177.928,6.291,148.526
C02512=1199.800,174.735,-55.840,-177.930,6.290,148.527
C02513=1199.805,174.486,-55.817,-177.933,6.288,148.527
C02514=1199.809,174.236,-55.795,-177.936,6.287,148.528
C02515=1199.814,173.988,-55.773,-177.938,6.285,148.528
C02516=1199.819,173.739,-55.750,-177.941,6.283,148.528
C02517=1199.823,173.489,-55.727,-177.944,6.281,148.529
C02518=1199.828,173.241,-55.706,-177.946,6.279,148.529
C02519=1199.833,172.992,-55.682,-177.948,6.278,148.529
C02520=1199.837,172.743,-55.661,-177.951,6.277,148.530
C02521=1199.842,172.494,-55.639,-177.954,6.275,148.530
C02522=1199.847,172.245,-55.616,-177.956,6.273,148.531
C02523=1199.851,171.996,-55.594,-177.959,6.271,148.531
C02524=1199.856,171.747,-55.572,-177.962,6.270,148.531
C02525=1199.860,171.498,-55.550,-177.964,6.269,148.532
C02526=1199.865,171.249,-55.527,-177.967,6.267,148.532
C02527=1199.870,171.000,-55.505,-177.970,6.265,148.533
C02528=1199.874,170.751,-55.483,-177.972,6.263,148.533
C02529=1199.879,170.503,-55.461,-177.975,6.262,148.533
C02530=1199.884,170.253,-55.439,-177.978,6.260,148.534
C02531=1199.889,170.005,-55.416,-177.980,6.258,148.534
C02532=1199.893,169.755,-55.394,-177.982,6.257,148.534
C02533=1199.898,169.507,-55.372,-177.985,6.255,148.535
C02534=1199.903,169.257,-55.350,-177.988,6.254,148.535
C02535=1199.908,169.009,-55.328,-177.991,6.252,148.536
C02536=1199.912,168.759,-55.306,-177.994,6.250,148.536
C02537=1199.917,168.511,-55.284,-177.996,6.249,148.536
C02538=1199.921,168.262,-55.262,-177.998,6.247,148.537
C02539=1199.926,168.013,-55.239,-178.001,6.246,148.537
C02540=1199.931,167.764,-55.217,-178.004,6.244,148.538
C02541=1199.936,167.515,-55.196,-178.006,6.242,148.538
C02542=1199.940,167.266,-55.174,-178.010,6.241,148.539
C02543=1199.945,167.017,-55.152,-178.012,6.240,148.539
C02544=1199.949,166.768,-55.130,-178.014,6.238,148.539
C02545=1199.954,166.519,-55.108,-178.017,6.236,148.540
C02546=1199.959,166.269,-55.085,-178.020,6.234,148.540
C02547=1199.964,166.021,-55.064,-178.022,6.232,148.540
C02548=1199.968,165.771,-55.042,-178.024,6.231,148.541
C02549=1199.973,165.523,-55.020,-178.027,6.230,148.541
C02550=1199.977,165.273,-54.998,-178.030,6.228,148.542
C02551=1199.982,165.025,-54.976,-178.033,6.226,148.542
C02552=1199.986,164.775,-54.954,-178.036,6.225,148.542
C02553=1199.991,164.527,-54.933,-178.038,6.224,148.543
C02554=1199.996,164.278,-54.911,-178.040,6.222,148.543
C02555=1200.000,164.029,-54.889,-178.043,6.220,148.544
C02556=1200.005,163.780,-54.867,-178.046,6.218,148.544
C02557=1200.009,163.531,-54.845,-178.049,6.217,148.545
C02558=1200.014,163.282,-54.823,-178.051,6.216,148.545
C02559=1200.019,163.032,-54.802,-178.054,6.214,148.545
C02560=1200.024,162.783,-54.780,-178.056,6.212,148.546
C02561=1200.029,162.535,-54.758,-178.059,6.210,148.546
C02562=1200.034,162.285,-54.736,-178.062,6.209,148.546
C02563=1200.038,162.037,-54.714,-178.064,6.208,148.547
C02564=1200.043,161.787,-54.692,-178.067,6.206,148.547
C02565=1200.048,161.538,-54.671,-178.070,6.204,148.548
C02566=1200.052,161.290,-54.650,-178.072,6.203,148.548
C02567=1200.056,161.040,-54.628,-178.074,6.202,148.549
C02568=1200.061,160.792,-54.607,-178.077,6.200,148.549
C02569=1200.066,160.543,-54.585,-178.080,6.198,148.549
C02570=1200.071,160.293,-54.564,-178.083,6.197,148.550
C02571=1200.075,160.044,-54.542,-178.085,6.196,148.550
C02572=1200.080,159.796,-54.520,-178.088,6.194,148.551
C02573=1200.085,159.546,-54.498,-178.090,6.192,148.551
C02574=1200.090,159.277,-54.475,-178.093,6.190,148.551
C02575=1200.095,159.008,-54.452,-178.096,6.189,148.552
C02576=1200.100,158.739,-54.428,-178.099,6.187,148.552
C02577=1200.105,158.470,-54.405,-178.102,6.186,148.553
C02578=1200.110,158.222,-54.384,-178.105,6.184,148.553
C02579=1200.115,157.972,-54.363,-178.107,6.183,148.554
C02580=1200.119,157.723,-54.340,-178.109,6.181,148.554
C02581=1200.124,157.474,-54.319,-178.112,6.179,148.554
C02582=1200.129,157.225,-54.298,-178.115,6.178,148.555
C02583=1200.134,156.976,-54.276,-178.117,6.177,148.555
C02584=1200.138,156.727,-54.255,-178.120,6.175,148.556
C02585=1200.143,156.478,-54.234,-178.123,6.173,148.556
C02586=1200.148,156.230,-54.212,-178.125,6.172,148.557
C02587=1200.152,155.980,-54.191,-178.128,6.171,148.557
C02588=1200.157,155.731,-54.169,-178.131,6.169,148.558
C02589=1200.162,155.482,-54.148,-178.133,6.167,148.558
C02590=1200.166,155.233,-54.127,-178.136,6.166,148.558
C02591=1200.171,154.983,-54.106,-178.138,6.165,148.559
C02592=1200.176,154.735,-54.084,-178.141,6.163,148.559
C02593=1200.181,154.486,-54.062,-178.144,6.161,148.560
C02594=1200.186,154.237,-54.041,-178.147,6.160,148.560
C02595=1200.189,153.988,-54.020,-178.149,6.159,148.560
C02596=1200.194,153.739,-53.999,-178.151,6.157,148.561
C02597=1200.200,153.489,-53.978,-178.154,6.155,148.561
C02598=1200.205,153.241,-53.956,-178.157,6.154,148.562
C02599=1200.208,152.991,-53.936,-178.159,6.153,148.562
C02600=1200.213,152.742,-53.914,-178.162,6.151,148.563
C02601=1200.218,152.493,-53.893,-178.165,6.149,148.563
C02602=1200.223,152.244,-53.871,-178.167,6.148,148.564
C02603=1200.228,151.996,-53.851,-178.170,6.147,148.564
C02604=1200.232,151.746,-53.829,-178.173,6.145,148.564
C02605=1200.237,151.497,-53.808,-178.175,6.144,148.565
C02606=1200.242,151.248,-53.787,-178.177,6.142,148.565
C02607=1200.246,150.999,-53.766,-178.181,6.141,148.566
C02608=1200.252,150.750,-53.745,-178.183,6.139,148.566
C02609=1200.255,150.500,-53.724,-178.185,6.138,148.566
C02610=1200.260,150.252,-53.702,-178.188,6.136,148.567
C02611=1200.266,150.003,-53.681,-178.191,6.135,148.567
C02612=1200.270,149.754,-53.660,-178.193,6.134,148.568
C02613=1200.275,149.505,-53.639,-178.196,6.132,148.568
C02614=1200.280,149.256,-53.618,-178.199,6.130,148.569
C02615=1200.284,149.006,-53.598,-178.201,6.130,148.569
C02616=1200.289,148.757,-53.576,-178.204,6.128,148.570
C02617=1200.294,148.508,-53.555,-178.207,6.126,148.570
C02618=1200.298,148.259,-53.535,-178.209,6.124,148.570
C02619=1200.303,148.011,-53.513,-178.212,6.124,148.571
C02620=1200.308,147.762,-53.493,-178.215,6.122,148.571
C02621=1200.313,147.512,-53.472,-178.217,6.120,148.572
C02622=1200.317,147.262,-53.450,-178.219,6.119,148.572
C02623=1200.322,147.013,-53.430,-178.223,6.118,148.573
C02624=1200.327,146.765,-53.408,-178.225,6.116,148.573
C02625=1200.331,146.516,-53.388,-178.227,6.115,148.573
C02626=1200.336,146.267,-53.367,-178.230,6.113,148.574
C02627=1200.341,146.018,-53.346,-178.233,6.112,148.574
C02628=1200.346,145.768,-53.326,-178.235,6.111,148.575
C02629=1200.350,145.520,-53.304,-178.238,6.109,148.575
C02630=1200.355,145.271,-53.283,-178.241,6.107,148.576
C02631=1200.360,145.021,-53.262,-178.243,6.107,148.576
C02632=1200.364,144.772,-53.242,-178.246,6.105,148.577
C02633=1200.369,144.523,-53.221,-178.249,6.103,148.577
C02634=1200.374,144.274,-53.200,-178.251,6.102,148.577
C02635=1200.379,144.024,-53.179,-178.254,6.101,148.578
C02636=1200.383,143.775,-53.159,-178.257,6.099,148.578
C02637=1200.388,143.527,-53.139,-178.259,6.098,148.579
C02638=1200.393,143.278,-53.117,-178.262,6.096,148.579
C02639=1200.397,143.029,-53.097,-178.265,6.095,148.580
C02640=1200.402,142.780,-53.076,-178.267,6.094,148.580
C02641=1200.407,142.531,-53.055,-178.269,6.092,148.581
C02642=1200.412,142.281,-53.034,-178.273,6.090,148.581
C02643=1200.416,142.033,-53.014,-178.275,6.089,148.582
C02644=1200.422,141.783,-52.993,-178.277,6.088,148.582
C02645=1200.426,141.534,-52.973,-178.280,6.086,148.582
C02646=1200.430,141.285,-52.952,-178.283,6.085,148.583
C02647=1200.436,141.036,-52.931,-178.285,6.084,148.583
C02648=1200.440,140.787,-52.911,-178.287,6.083,148.584
C02649=1200.445,140.538,-52.890,-178.291,6.081,148.584
C02650=1200.450,140.289,-52.870,-178.293,6.079,148.585
C02651=1200.454,140.039,-52.850,-178.295,6.078,148.585
C02652=1200.460,139.790,-52.829,-178.299,6.077,148.586
C02653=1200.464,139.541,-52.809,-178.301,6.075,148.586
C02654=1200.469,139.292,-52.788,-178.303,6.074,148.587
C02655=1200.474,139.043,-52.767,-178.306,6.072,148.587
C02656=1200.478,138.794,-52.747,-178.309,6.071,148.588
C02657=1200.483,138.545,-52.726,-178.311,6.070,148.588
C02658=1200.488,138.296,-52.706,-178.314,6.068,148.588
C02659=1200.492,138.047,-52.685,-178.317,6.068,148.589
C02660=1200.498,137.797,-52.665,-178.319,6.066,148.589
C02661=1200.502,137.548,-52.645,-178.322,6.064,148.590
C02662=1200.506,137.299,-52.624,-178.325,6.064,148.590
C02663=1200.511,137.050,-52.604,-178.327,6.062,148.591
C02664=1200.516,136.801,-52.583,-178.330,6.060,148.591
C02665=1200.521,136.551,-52.563,-178.333,6.059,148.592
C02666=1200.525,136.302,-52.543,-178.335,6.058,148.592
C02667=1200.530,136.053,-52.522,-178.337,6.057,148.593
C02668=1200.535,135.804,-52.501,-178.340,6.055,148.593
C02669=1200.540,135.555,-52.482,-178.343,6.053,148.594
C02670=1200.544,135.306,-52.461,-178.345,6.052,148.594
C02671=1200.549,135.056,-52.440,-178.348,6.051,148.594
C02672=1200.554,134.808,-52.420,-178.351,6.050,148.595
C02673=1200.559,134.559,-52.401,-178.353,6.048,148.595
C02674=1200.563,134.310,-52.380,-178.356,6.047,148.596
C02675=1200.569,134.060,-52.359,-178.359,6.046,148.596
C02676=1200.573,133.811,-52.340,-178.361,6.044,148.597
C02677=1200.578,133.562,-52.319,-178.363,6.043,148.597
C02678=1200.583,133.293,-52.297,-178.367,6.042,148.598
C02679=1200.588,133.025,-52.276,-178.369,6.040,148.598
C02680=1200.594,132.756,-52.254,-178.372,6.039,148.599
C02681=1200.598,132.488,-52.232,-178.376,6.037,148.599
C02682=1200.603,132.238,-52.213,-178.378,6.036,148.600
C02683=1200.608,131.989,-52.192,-178.380,6.034,148.600
C02684=1200.613,131.740,-52.171,-178.383,6.034,148.601
C02685=1200.617,131.490,-52.152,-178.386,6.032,148.601
C02686=1200.622,131.242,-52.132,-178.388,6.031,148.602
C02687=1200.627,130.993,-52.112,-178.391,6.030,148.602
C02688=1200.632,130.744,-52.092,-178.394,6.028,148.603
C02689=1200.636,130.494,-52.072,-178.396,6.027,148.603
C02690=1200.642,130.245,-52.051,-178.399,6.026,148.604
C02691=1200.646,129.996,-52.031,-178.401,6.025,148.604
C02692=1200.651,129.747,-52.012,-178.404,6.023,148.604
C02693=1200.656,129.498,-51.991,-178.406,6.022,148.605
C02694=1200.661,129.249,-51.971,-178.409,6.020,148.605
C02695=1200.665,129.000,-51.951,-178.412,6.019,148.606
C02696=1200.670,128.750,-51.931,-178.414,6.018,148.606
C02697=1200.675,128.502,-51.911,-178.417,6.016,148.607
C02698=1200.680,128.252,-51.892,-178.420,6.016,148.607
C02699=1200.684,128.003,-51.872,-178.422,6.014,148.608
C02700=1200.689,127.754,-51.852,-178.424,6.013,148.608
C02701=1200.693,127.504,-51.832,-178.428,6.012,148.609
C02702=1200.698,127.256,-51.812,-178.430,6.010,148.609
C02703=1200.703,127.006,-51.792,-178.432,6.009,148.610
C02704=1200.708,126.757,-51.772,-178.436,6.007,148.610
C02705=1200.712,126.508,-51.752,-178.438,6.006,148.611
C02706=1200.717,126.258,-51.733,-178.440,6.005,148.611
C02707=1200.722,126.010,-51.713,-178.443,6.004,148.612
C02708=1200.727,125.760,-51.693,-178.446,6.002,148.612
C02709=1200.732,125.511,-51.673,-178.448,6.002,148.613
C02710=1200.736,125.262,-51.653,-178.451,6.000,148.613
C02711=1200.741,125.013,-51.634,-178.453,5.999,148.614
C02712=1200.746,124.763,-51.614,-178.456,5.998,148.614
C02713=1200.751,124.515,-51.594,-178.459,5.996,148.615
C02714=1200.756,124.266,-51.574,-178.462,5.995,148.615
C02715=1200.761,124.016,-51.555,-178.464,5.993,148.616
C02716=1200.765,123.767,-51.534,-178.466,5.993,148.616
C02717=1200.770,123.518,-51.515,-178.470,5.991,148.617
C02718=1200.775,123.269,-51.495,-178.472,5.990,148.617
C02719=1200.780,123.019,-51.476,-178.475,5.989,148.618
C02720=1200.784,122.770,-51.455,-178.477,5.988,148.618
C02721=1200.790,122.521,-51.436,-178.480,5.986,148.618
C02722=1200.794,122.272,-51.417,-178.482,5.985,148.619
C02723=1200.799,122.022,-51.397,-178.485,5.984,148.619
C02724=1200.804,121.774,-51.378,-178.487,5.983,148.620
C02725=1200.808,121.525,-51.358,-178.490,5.981,148.621
C02726=1200.813,121.275,-51.338,-178.492,5.980,148.621
C02727=1200.818,121.026,-51.319,-178.496,5.979,148.622
C02728=1200.823,120.777,-51.299,-178.498,5.978,148.622
C02729=1200.828,120.527,-51.280,-178.501,5.977,148.623
C02730=1200.832,120.279,-51.261,-178.503,5.976,148.623
C02731=1200.837,120.030,-51.240,-178.506,5.974,148.623
C02732=1200.842,119.780,-51.221,-178.508,5.973,148.624
C02733=1200.847,119.531,-51.202,-178.511,5.972,148.624
C02734=1200.852,119.282,-51.182,-178.514,5.971,148.625
C02735=1200.856,119.032,-51.162,-178.516,5.969,148.625
C02736=1200.861,118.783,-51.144,-178.518,5.968,148.626
C02737=1200.866,118.534,-51.124,-178.522,5.967,148.626
C02738=1200.871,118.284,-51.104,-178.524,5.966,148.627
C02739=1200.876,118.035,-51.085,-178.527,5.964,148.628
C02740=1200.880,117.786,-51.066,-178.529,5.964,148.628
C02741=1200.885,117.537,-51.047,-178.532,5.962,148.629
C02742=1200.890,117.288,-51.027,-178.534,5.961,148.629
C02743=1200.895,117.038,-51.007,-178.537,5.959,148.629
C02744=1200.900,116.789,-50.988,-178.540,5.959,148.630
C02745=1200.904,116.540,-50.969,-178.542,5.957,148.630
C02746=1200.909,116.291,-50.950,-178.545,5.956,148.631
C02747=1200.914,116.042,-50.930,-178.548,5.955,148.631
C02748=1200.919,115.793,-50.911,-178.550,5.954,148.632
C02749=1200.924,115.544,-50.892,-178.553,5.952,148.632
C02750=1200.928,115.294,-50.872,-178.555,5.951,148.633
C02751=1200.934,115.045,-50.853,-178.558,5.950,148.634
C02752=1200.938,114.796,-50.834,-178.560,5.949,148.634
C02753=1200.943,114.547,-50.814,-178.564,5.948,148.635
C02754=1200.948,114.297,-50.795,-178.566,5.947,148.635
C02755=1200.952,114.049,-50.776,-178.569,5.945,148.636
C02756=1200.957,113.799,-50.756,-178.571,5.944,148.636
C02757=1200.962,113.550,-50.737,-178.574,5.943,148.637
C02758=1200.967,113.301,-50.719,-178.576,5.942,148.637
C02759=1200.972,113.052,-50.699,-178.579,5.940,148.637
C02760=1200.977,112.802,-50.680,-178.582,5.940,148.638
C02761=1200.981,112.553,-50.661,-178.584,5.938,148.638
C02762=1200.986,112.304,-50.641,-178.587,5.937,148.639
C02763=1200.991,112.054,-50.622,-178.589,5.936,148.640
C02764=1200.996,111.805,-50.604,-178.592,5.935,148.640
C02765=1201.001,111.556,-50.584,-178.594,5.934,148.641
C02766=1201.005,111.307,-50.565,-178.598,5.933,148.641
C02767=1201.010,111.058,-50.546,-178.600,5.932,148.642
C02768=1201.015,110.809,-50.526,-178.603,5.930,148.642
C02769=1201.020,110.559,-50.508,-178.605,5.929,148.643
C02770=1201.025,110.310,-50.489,-178.608,5.928,148.643
C02771=1201.029,110.061,-50.470,-178.610,5.927,148.644
C02772=1201.034,109.812,-50.450,-178.613,5.925,148.644
C02773=1201.039,109.563,-50.432,-178.616,5.925,148.645
C02774=1201.044,109.313,-50.413,-178.618,5.924,148.645
C02775=1201.049,109.064,-50.394,-178.621,5.922,148.646
C02776=1201.054,108.814,-50.375,-178.623,5.921,148.646
C02777=1201.059,108.565,-50.356,-178.626,5.920,148.647
C02778=1201.063,108.316,-50.337,-178.628,5.919,148.647
C02779=1201.069,108.067,-50.318,-178.632,5.918,148.648
C02780=1201.073,107.817,-50.299,-178.634,5.917,148.648
C02781=1201.078,107.569,-50.280,-178.636,5.916,148.649
C02782=1201.083,107.300,-50.260,-178.639,5.914,148.649
C02783=1201.088,107.032,-50.239,-178.642,5.913,148.650
C02784=1201.094,106.763,-50.219,-178.645,5.912,148.651
C02785=1201.098,106.495,-50.199,-178.648,5.911,148.651
C02786=1201.104,106.245,-50.180,-178.650,5.910,148.652
C02787=1201.108,105.997,-50.162,-178.653,5.908,148.652
C02788=1201.113,105.747,-50.142,-178.655,5.908,148.653
C02789=1201.118,105.498,-50.124,-178.658,5.906,148.653
C02790=1201.123,105.248,-50.104,-178.661,5.905,148.654
C02791=1201.127,104.999,-50.086,-178.663,5.904,148.654
C02792=1201.133,104.750,-50.067,-178.666,5.903,148.655
C02793=1201.137,104.500,-50.049,-178.668,5.902,148.655
C02794=1201.142,104.252,-50.030,-178.671,5.901,148.656
C02795=1201.147,104.002,-50.011,-178.674,5.900,148.656
C02796=1201.151,103.753,-49.992,-178.676,5.899,148.657
C02797=1201.157,103.504,-49.974,-178.679,5.897,148.657
C02798=1201.161,103.254,-49.955,-178.681,5.897,148.658
C02799=1201.166,103.005,-49.937,-178.684,5.895,148.658
C02800=1201.171,102.756,-49.917,-178.687,5.895,148.659
C02801=1201.176,102.507,-49.899,-178.690,5.893,148.659
C02802=1201.180,102.258,-49.880,-178.692,5.892,148.660
C02803=1201.186,102.008,-49.862,-178.694,5.891,148.660
C02804=1201.190,101.759,-49.844,-178.697,5.890,148.661
C02805=1201.196,101.510,-49.824,-178.700,5.889,148.662
C02806=1201.200,101.261,-49.806,-178.703,5.888,148.662
C02807=1201.204,101.011,-49.787,-178.705,5.887,148.663
C02808=1201.209,100.762,-49.769,-178.708,5.886,148.663
C02809=1201.215,100.513,-49.751,-178.710,5.884,148.664
C02810=1201.219,100.263,-49.732,-178.713,5.884,148.664
C02811=1201.224,100.014,-49.714,-178.715,5.883,148.665
C02812=1201.229,99.765,-49.694,-178.718,5.881,148.665
C02813=1201.234,99.515,-49.676,-178.720,5.880,148.666
C02814=1201.238,99.266,-49.658,-178.723,5.879,148.666
C02815=1201.244,99.017,-49.639,-178.726,5.878,148.667
C02816=1201.248,98.768,-49.620,-178.728,5.878,148.667
C02817=1201.253,98.518,-49.602,-178.731,5.876,148.668
C02818=1201.258,98.269,-49.584,-178.734,5.875,148.669
C02819=1201.263,98.020,-49.565,-178.736,5.875,148.669
C02820=1201.268,97.770,-49.547,-178.739,5.873,148.670
C02821=1201.273,97.521,-49.529,-178.741,5.872,148.670
C02822=1201.277,97.273,-49.510,-178.744,5.871,148.671
C02823=1201.283,97.023,-49.491,-178.747,5.870,148.671
C02824=1201.287,96.773,-49.473,-178.749,5.869,148.672
C02825=1201.292,96.524,-49.455,-178.752,5.868,148.672
C02826=1201.297,96.275,-49.437,-178.754,5.867,148.673
C02827=1201.302,96.026,-49.418,-178.757,5.866,148.673
C02828=1201.307,95.776,-49.400,-178.760,5.864,148.674
C02829=1201.311,95.527,-49.382,-178.762,5.864,148.674
C02830=1201.316,95.278,-49.364,-178.765,5.862,148.675
C02831=1201.321,95.029,-49.346,-178.768,5.861,148.676
C02832=1201.325,94.779,-49.327,-178.770,5.861,148.676
C02833=1201.330,94.530,-49.309,-178.773,5.859,148.677
C02834=1201.336,94.281,-49.290,-178.775,5.859,148.677
C02835=1201.341,94.032,-49.272,-178.778,5.858,148.678
C02836=1201.346,93.782,-49.254,-178.781,5.856,148.678
C02837=1201.350,93.533,-49.236,-178.783,5.855,148.679
C02838=1201.355,93.283,-49.218,-178.786,5.855,148.679
C02839=1201.360,93.034,-49.200,-178.788,5.853,148.680
C02840=1201.365,92.785,-49.182,-178.791,5.852,148.680
C02841=1201.370,92.536,-49.162,-178.793,5.852,148.681
C02842=1201.374,92.286,-49.144,-178.796,5.850,148.682
C02843=1201.379,92.037,-49.126,-178.799,5.850,148.682
C02844=1201.384,91.788,-49.108,-178.801,5.849,148.683
C02845=1201.389,91.539,-49.090,-178.804,5.847,148.683
C02846=1201.394,91.290,-49.072,-178.806,5.846,148.684
C02847=1201.399,91.040,-49.054,-178.809,5.846,148.684
C02848=1201.403,90.791,-49.036,-178.812,5.844,148.685
C02849=1201.408,90.541,-49.018,-178.814,5.843,148.685
C02850=1201.413,90.292,-49.000,-178.817,5.843,148.686
C02851=1201.418,90.043,-48.982,-178.820,5.841,148.686
C02852=1201.423,89.794,-48.964,-178.822,5.841,148.687
C02853=1201.428,89.545,-48.946,-178.824,5.840,148.688
C02854=1201.433,89.296,-48.928,-178.828,5.838,148.688
C02855=1201.437,89.046,-48.910,-178.830,5.837,148.689
C02856=1201.442,88.796,-48.892,-178.832,5.837,148.689
C02857=1201.447,88.547,-48.874,-178.835,5.835,148.690
C02858=1201.452,88.297,-48.856,-178.838,5.834,148.690
C02859=1201.457,88.048,-48.838,-178.840,5.834,148.691
C02860=1201.462,87.799,-48.820,-178.843,5.832,148.691
C02861=1201.467,87.550,-48.802,-178.846,5.832,148.692
C02862=1201.472,87.301,-48.784,-178.848,5.831,148.692
C02863=1201.477,87.052,-48.767,-178.851,5.829,148.693
C02864=1201.482,86.802,-48.749,-178.854,5.829,148.694
C02865=1201.486,86.553,-48.730,-178.856,5.828,148.694
C02866=1201.491,86.303,-48.713,-178.858,5.827,148.695
C02867=1201.496,86.054,-48.695,-178.861,5.825,148.695
C02868=1201.501,85.804,-48.677,-178.864,5.825,148.696
C02869=1201.506,85.555,-48.659,-178.866,5.824,148.696
C02870=1201.511,85.306,-48.641,-178.869,5.823,148.697
C02871=1201.516,85.057,-48.623,-178.872,5.822,148.698
C02872=1201.521,84.807,-48.606,-178.874,5.821,148.698
C02873=1201.526,84.558,-48.588,-178.877,5.820,148.699
C02874=1201.531,84.309,-48.570,-178.879,5.819,148.699
C02875=1201.535,84.060,-48.552,-178.882,5.818,148.700
C02876=1201.540,83.810,-48.535,-178.884,5.818,148.700
C02877=1201.545,83.561,-48.517,-178.887,5.816,148.701
C02878=1201.550,83.312,-48.499,-178.890,5.815,148.701
C02879=1201.555,83.063,-48.481,-178.892,5.814,148.702
C02880=1201.560,82.813,-48.464,-178.895,5.813,148.703
C02881=1201.565,82.564,-48.446,-178.898,5.812,148.703
C02882=1201.569,82.315,-48.429,-178.900,5.812,148.704
C02883=1201.574,82.065,-48.411,-178.902,5.811,148.704
C02884=1201.579,81.816,-48.393,-178.905,5.809,148.705
C02885=1201.584,81.567,-48.375,-178.908,5.809,148.705
C02886=1201.590,81.298,-48.357,-178.910,5.808,148.706
C02887=1201.595,81.029,-48.337,-178.914,5.807,148.707
C02888=1201.600,80.761,-48.319,-178.916,5.806,148.707
C02889=1201.605,80.492,-48.299,-178.919,5.804,148.708
C02890=1201.610,80.243,-48.282,-178.921,5.804,148.708
C02891=1201.614,79.994,-48.265,-178.924,5.803,148.709
C02892=1201.619,79.744,-48.247,-178.927,5.802,148.709
C02893=1201.625,79.495,-48.229,-178.929,5.801,148.710
C02894=1201.630,79.245,-48.211,-178.932,5.800,148.711
C02895=1201.634,78.996,-48.195,-178.934,5.800,148.711
C02896=1201.640,78.748,-48.177,-178.937,5.798,148.712
C02897=1201.644,78.498,-48.159,-178.940,5.797,148.712
C02898=1201.650,78.249,-48.142,-178.942,5.797,148.713
C02899=1201.654,78.000,-48.124,-178.944,5.796,148.713
C02900=1201.659,77.750,-48.107,-178.948,5.794,148.714
C02901=1201.664,77.501,-48.089,-178.950,5.794,148.715
C02902=1201.668,77.251,-48.072,-178.952,5.793,148.715
C02903=1201.673,77.002,-48.054,-178.955,5.792,148.716
C02904=1201.679,76.752,-48.037,-178.958,5.791,148.716
C02905=1201.683,76.503,-48.019,-178.960,5.790,148.717
C02906=1201.688,76.254,-48.003,-178.963,5.790,148.718
C02907=1201.693,76.004,-47.985,-178.965,5.789,148.718
C02908=1201.698,75.755,-47.967,-178.968,5.787,148.719
C02909=1201.702,75.506,-47.950,-178.971,5.787,148.719
C02910=1201.708,75.257,-47.933,-178.973,5.786,148.720
C02911=1201.713,75.007,-47.916,-178.976,5.785,148.720
C02912=1201.717,74.758,-47.898,-178.979,5.784,148.721
C02913=1201.723,74.508,-47.881,-178.981,5.783,148.721
C02914=1201.728,74.259,-47.863,-178.984,5.782,148.722
C02915=1201.732,74.010,-47.846,-178.986,5.782,148.723
C02916=1201.737,73.760,-47.829,-178.989,5.780,148.723
C02917=1201.741,73.511,-47.812,-178.992,5.780,148.724
C02918=1201.747,73.262,-47.795,-178.994,5.779,148.724
C02919=1201.753,73.012,-47.778,-178.996,5.778,148.725
C02920=1201.757,72.763,-47.760,-178.999,5.777,148.726
C02921=1201.762,72.513,-47.743,-179.002,5.776,148.726
C02922=1201.766,72.264,-47.726,-179.004,5.775,148.727
C02923=1201.771,72.015,-47.708,-179.007,5.775,148.727
C02924=1201.777,71.765,-47.691,-179.009,5.774,148.728
C02925=1201.782,71.516,-47.675,-179.012,5.772,148.728
C02926=1201.787,71.267,-47.657,-179.015,5.772,148.729
C02927=1201.791,71.017,-47.640,-179.017,5.771,148.729
C02928=1201.796,70.768,-47.623,-179.020,5.770,148.730
C02929=1201.800,70.519,-47.605,-179.022,5.770,148.731
C02930=1201.806,70.269,-47.588,-179.025,5.768,148.731
C02931=1201.811,70.020,-47.571,-179.028,5.767,148.732
C02932=1201.816,69.770,-47.555,-179.030,5.767,148.733
C02933=1201.821,69.521,-47.537,-179.032,5.766,148.733
C02934=1201.825,69.272,-47.520,-179.036,5.765,148.734
C02935=1201.831,69.022,-47.503,-179.038,5.764,148.734
C02936=1201.836,68.773,-47.486,-179.040,5.763,148.735
C02937=1201.841,68.523,-47.469,-179.043,5.763,148.735
C02938=1201.845,68.275,-47.452,-179.045,5.762,148.736
C02939=1201.850,68.025,-47.435,-179.048,5.760,148.736
C02940=1201.855,67.775,-47.418,-179.051,5.760,148.737
C02941=1201.860,67.526,-47.402,-179.053,5.759,148.738
C02942=1201.865,67.277,-47.384,-179.056,5.758,148.738
C02943=1201.869,67.027,-47.368,-179.058,5.758,148.739
C02944=1201.875,66.777,-47.350,-179.061,5.756,148.739
C02945=1201.879,66.529,-47.333,-179.064,5.756,148.740
C02946=1201.885,66.279,-47.316,-179.066,5.755,148.741
C02947=1201.889,66.030,-47.299,-179.069,5.754,148.741
C02948=1201.894,65.780,-47.282,-179.071,5.754,148.742
C02949=1201.899,65.531,-47.266,-179.074,5.753,148.742
C02950=1201.904,65.282,-47.249,-179.077,5.751,148.743
C02951=1201.909,65.032,-47.232,-179.079,5.751,148.743
C02952=1201.914,64.783,-47.215,-179.082,5.750,148.744
C02953=1201.919,64.534,-47.198,-179.084,5.749,148.745
C02954=1201.924,64.284,-47.182,-179.087,5.749,148.745
C02955=1201.928,64.035,-47.165,-179.090,5.747,148.746
C02956=1201.934,63.785,-47.148,-179.092,5.747,148.747
C02957=1201.939,63.536,-47.131,-179.095,5.746,148.747
C02958=1201.943,63.286,-47.115,-179.097,5.745,148.748
C02959=1201.948,63.037,-47.098,-179.100,5.745,148.748
C02960=1201.953,62.788,-47.081,-179.102,5.744,148.749
C02961=1201.959,62.538,-47.064,-179.105,5.742,148.749
C02962=1201.963,62.289,-47.047,-179.108,5.742,148.750
C02963=1201.968,62.040,-47.031,-179.110,5.741,148.751
C02964=1201.973,61.790,-47.014,-179.113,5.740,148.751
C02965=1201.978,61.541,-46.997,-179.115,5.740,148.752
C02966=1201.983,61.292,-46.981,-179.117,5.739,148.752
C02967=1201.988,61.042,-46.963,-179.121,5.738,148.753
C02968=1201.993,60.793,-46.947,-179.123,5.737,148.754
C02969=1201.998,60.544,-46.930,-179.125,5.736,148.754
C02970=1202.002,60.294,-46.914,-179.128,5.736,148.755
C02971=1202.008,60.044,-46.897,-179.131,5.735,148.755
C02972=1202.013,59.795,-46.881,-179.133,5.735,148.756
C02973=1202.017,59.546,-46.864,-179.136,5.733,148.756
C02974=1202.023,59.296,-46.847,-179.139,5.732,148.757
C02975=1202.028,59.047,-46.831,-179.141,5.732,148.758
C02976=1202.032,58.797,-46.814,-179.143,5.731,148.758
C02977=1202.037,58.549,-46.798,-179.146,5.730,148.759
C02978=1202.042,58.299,-46.780,-179.149,5.730,148.760
C02979=1202.047,58.049,-46.765,-179.151,5.729,148.760
C02980=1202.052,57.800,-46.748,-179.154,5.728,148.761
C02981=1202.057,57.551,-46.732,-179.157,5.727,148.761
C02982=1202.061,57.301,-46.715,-179.159,5.726,148.762
C02983=1202.067,57.052,-46.698,-179.161,5.726,148.762
C02984=1202.072,56.802,-46.682,-179.164,5.725,148.763
C02985=1202.077,56.553,-46.666,-179.167,5.724,148.764
C02986=1202.081,56.304,-46.649,-179.169,5.724,148.764
C02987=1202.087,56.055,-46.633,-179.172,5.722,148.765
C02988=1202.092,55.804,-46.616,-179.175,5.722,148.766
C02989=1202.097,55.555,-46.600,-179.177,5.721,148.766
C02990=1202.102,55.287,-46.582,-179.179,5.720,148.767
C02991=1202.107,55.019,-46.565,-179.182,5.720,148.767
C02992=1202.113,54.750,-46.546,-179.185,5.718,148.768
C02993=1202.118,54.481,-46.529,-179.188,5.718,148.769
C02994=1202.123,54.232,-46.512,-179.191,5.717,148.769
C02995=1202.128,53.983,-46.496,-179.193,5.717,148.770
C02996=1202.133,53.733,-46.480,-179.195,5.716,148.770
C02997=1202.138,53.484,-46.464,-179.199,5.714,148.771
C02998=1202.143,53.234,-46.448,-179.201,5.714,148.772
C02999=1202.148,52.985,-46.431,-179.203,5.713,148.772
C03000=1202.153,52.735,-46.414,-179.206,5.712,148.773
C03001=1202.158,52.486,-46.399,-179.209,5.712,148.774
C03002=1202.163,52.237,-46.382,-179.211,5.711,148.774
C03003=1202.167,51.987,-46.365,-179.213,5.710,148.775
C03004=1202.173,51.738,-46.350,-179.216,5.710,148.775
C03005=1202.177,51.488,-46.333,-179.219,5.709,148.776
C03006=1202.182,51.239,-46.318,-179.221,5.708,148.776
C03007=1202.187,50.989,-46.301,-179.224,5.707,148.777
C03008=1202.192,50.740,-46.285,-179.227,5.707,148.778
C03009=1202.197,50.490,-46.269,-179.229,5.706,148.778
C03010=1202.202,50.242,-46.252,-179.231,5.705,148.779
C03011=1202.207,49.991,-46.236,-179.234,5.705,148.780
C03012=1202.212,49.743,-46.220,-179.237,5.704,148.780
C03013=1202.216,49.493,-46.204,-179.239,5.704,148.781
C03014=1202.222,49.244,-46.188,-179.242,5.703,148.781
C03015=1202.226,48.994,-46.172,-179.244,5.702,148.782
C03016=1202.231,48.745,-46.156,-179.247,5.701,148.783
C03017=1202.237,48.496,-46.140,-179.250,5.700,148.783
C03018=1202.241,48.246,-46.123,-179.252,5.699,148.784
C03019=1202.247,47.997,-46.108,-179.255,5.699,148.784
C03020=1202.251,47.747,-46.091,-179.257,5.698,148.785
C03021=1202.257,47.498,-46.075,-179.260,5.697,148.786
C03022=1202.261,47.248,-46.060,-179.262,5.697,148.786
C03023=1202.266,46.999,-46.043,-179.265,5.696,148.787
C03024=1202.271,46.749,-46.027,-179.268,5.696,148.788
C03025=1202.276,46.500,-46.011,-179.270,5.695,148.788
C03026=1202.281,46.250,-45.995,-179.272,5.694,148.789
C03027=1202.286,46.001,-45.979,-179.276,5.693,148.789
C03028=1202.292,45.752,-45.963,-179.278,5.692,148.790
C03029=1202.296,45.502,-45.947,-179.280,5.692,148.790
C03030=1202.301,45.253,-45.931,-179.283,5.691,148.791
C03031=1202.306,45.003,-45.915,-179.286,5.690,148.792
C03032=1202.312,44.753,-45.899,-179.288,5.690,148.792
C03033=1202.317,44.505,-45.883,-179.290,5.689,148.793
C03034=1202.321,44.254,-45.867,-179.293,5.688,148.794
C03035=1202.326,44.005,-45.852,-179.296,5.688,148.794
C03036=1202.331,43.756,-45.835,-179.298,5.687,148.795
C03037=1202.336,43.506,-45.820,-179.300,5.687,148.795
C03038=1202.341,43.257,-45.804,-179.303,5.686,148.796
C03039=1202.346,43.008,-45.788,-179.306,5.685,148.797
C03040=1202.351,42.758,-45.772,-179.308,5.685,148.797
C03041=1202.356,42.508,-45.756,-179.311,5.683,148.798
C03042=1202.361,42.259,-45.740,-179.314,5.683,148.798
C03043=1202.366,42.010,-45.725,-179.316,5.682,148.799
C03044=1202.371,41.760,-45.709,-179.319,5.682,148.800
C03045=1202.376,41.511,-45.693,-179.321,5.681,148.800
C03046=1202.381,41.261,-45.678,-179.324,5.680,148.801
C03047=1202.386,41.012,-45.661,-179.326,5.680,148.802
C03048=1202.391,40.762,-45.645,-179.329,5.679,148.802
C03049=1202.396,40.513,-45.630,-179.331,5.678,148.803
C03050=1202.401,40.263,-45.614,-179.334,5.678,148.803
C03051=1202.406,40.014,-45.598,-179.337,5.677,148.804
C03052=1202.411,39.765,-45.582,-179.339,5.677,148.805
C03053=1202.416,39.515,-45.567,-179.341,5.676,148.805
C03054=1202.421,39.266,-45.552,-179.344,5.675,148.806
C03055=1202.426,39.016,-45.536,-179.347,5.675,148.807
C03056=1202.431,38.766,-45.520,-179.349,5.674,148.807
C03057=1202.436,38.517,-45.504,-179.351,5.673,148.808
C03058=1202.440,38.268,-45.489,-179.354,5.673,148.808
C03059=1202.445,38.018,-45.473,-179.357,5.672,148.809
C03060=1202.451,37.769,-45.457,-179.360,5.671,148.810
C03061=1202.456,37.519,-45.442,-179.363,5.670,148.810
C03062=1202.461,37.270,-45.427,-179.365,5.669,148.811
C03063=1202.465,37.020,-45.411,-179.367,5.669,148.811
C03064=1202.471,36.771,-45.395,-179.370,5.668,148.812
C03065=1202.476,36.521,-45.379,-179.373,5.668,148.813
C03066=1202.481,36.272,-45.364,-179.375,5.667,148.813
C03067=1202.486,36.022,-45.349,-179.377,5.666,148.814
C03068=1202.491,35.773,-45.333,-179.380,5.666,148.815
C03069=1202.496,35.524,-45.318,-179.383,5.665,148.815
C03070=1202.500,35.274,-45.302,-179.385,5.665,148.816
C03071=1202.506,35.025,-45.286,-179.387,5.664,148.816
C03072=1202.510,34.776,-45.271,-179.390,5.664,148.817
C03073=1202.516,34.526,-45.255,-179.393,5.663,148.818
C03074=1202.520,34.276,-45.239,-179.395,5.662,148.818
C03075=1202.525,34.027,-45.224,-179.398,5.662,148.819
C03076=1202.531,33.777,-45.209,-179.400,5.661,148.820
C03077=1202.536,33.528,-45.194,-179.403,5.661,148.820
C03078=1202.541,33.279,-45.179,-179.405,5.660,148.821
C03079=1202.546,33.029,-45.163,-179.408,5.659,148.821
C03080=1202.551,32.779,-45.147,-179.410,5.659,148.822
C03081=1202.556,32.530,-45.132,-179.413,5.658,148.823
C03082=1202.561,32.281,-45.117,-179.416,5.658,148.823
C03083=1202.565,32.031,-45.101,-179.418,5.657,148.824
C03084=1202.570,31.782,-45.086,-179.420,5.656,148.825
C03085=1202.576,31.532,-45.070,-179.423,5.656,148.825
C03086=1202.580,31.283,-45.055,-179.426,5.655,148.826
C03087=1202.586,31.034,-45.039,-179.428,5.655,148.827
C03088=1202.590,30.784,-45.024,-179.430,5.654,148.827
C03089=1202.596,30.534,-45.009,-179.433,5.653,148.828
C03090=1202.601,30.284,-44.994,-179.436,5.653,148.828
C03091=1202.606,30.035,-44.979,-179.438,5.652,148.829
C03092=1202.611,29.786,-44.963,-179.441,5.652,148.830
C03093=1202.616,29.537,-44.948,-179.443,5.651,148.830
C03094=1202.621,29.268,-44.932,-179.446,5.650,148.831
C03095=1202.626,28.999,-44.915,-179.448,5.650,148.832
C03096=1202.632,28.730,-44.899,-179.452,5.648,148.832
C03097=1202.637,28.461,-44.882,-179.454,5.648,148.833
C03098=1202.642,28.212,-44.867,-179.457,5.647,148.834
C03099=1202.647,27.962,-44.852,-179.460,5.647,148.834
C03100=1202.652,27.713,-44.837,-179.462,5.646,148.835
C03101=1202.657,27.464,-44.821,-179.465,5.646,148.836
C03102=1202.662,27.215,-44.806,-179.467,5.645,148.836
C03103=1202.668,26.965,-44.791,-179.470,5.644,148.837
C03104=1202.672,26.715,-44.776,-179.472,5.644,148.837
C03105=1202.677,26.465,-44.760,-179.475,5.643,148.838
C03106=1202.682,26.216,-44.746,-179.478,5.643,148.839
C03107=1202.688,25.966,-44.731,-179.480,5.642,148.839
C03108=1202.692,25.717,-44.716,-179.482,5.641,148.840
C03109=1202.697,25.468,-44.701,-179.485,5.641,148.841
C03110=1202.703,25.218,-44.686,-179.488,5.640,148.841
C03111=1202.707,24.969,-44.671,-179.490,5.640,148.842
C03112=1202.713,24.720,-44.655,-179.492,5.640,148.842
C03113=1202.717,24.469,-44.640,-179.495,5.639,148.843
C03114=1202.722,24.220,-44.625,-179.497,5.639,148.844
C03115=1202.727,23.971,-44.610,-179.500,5.638,148.844
C03116=1202.732,23.721,-44.596,-179.503,5.638,148.845
C03117=1202.737,23.472,-44.580,-179.505,5.637,148.846
C03118=1202.742,23.222,-44.565,-179.507,5.636,148.846
C03119=1202.748,22.972,-44.550,-179.510,5.636,148.847
C03120=1202.752,22.723,-44.535,-179.513,5.635,148.848
C03121=1202.757,22.474,-44.521,-179.515,5.635,148.848
C03122=1202.763,22.224,-44.505,-179.517,5.634,148.849
C03123=1202.767,21.975,-44.490,-179.520,5.633,148.849
C03124=1202.773,21.725,-44.475,-179.523,5.633,148.850
C03125=1202.778,21.476,-44.460,-179.525,5.632,148.851
C03126=1202.783,21.226,-44.446,-179.528,5.632,148.851
C03127=1202.788,20.977,-44.431,-179.530,5.631,148.852
C03128=1202.793,20.727,-44.416,-179.533,5.630,148.853
C03129=1202.797,20.477,-44.401,-179.536,5.630,148.853
C03130=1202.803,20.227,-44.386,-179.538,5.629,148.854
C03131=1202.807,19.978,-44.371,-179.541,5.629,148.855
C03132=1202.812,19.729,-44.357,-179.543,5.628,148.855
C03133=1202.818,19.479,-44.341,-179.546,5.628,148.856
C03134=1202.823,19.229,-44.327,-179.548,5.627,148.856
C03135=1202.827,18.980,-44.312,-179.551,5.626,148.857
C03136=1202.832,18.731,-44.298,-179.554,5.626,148.858
C03137=1202.838,18.481,-44.282,-179.556,5.626,148.858
C03138=1202.843,18.232,-44.268,-179.558,5.625,148.859
C03139=1202.847,17.982,-44.253,-179.560,5.625,148.860
C03140=1202.853,17.732,-44.238,-179.563,5.624,148.860
C03141=1202.858,17.483,-44.223,-179.566,5.624,148.861
C03142=1202.863,17.234,-44.209,-179.568,5.623,148.862
C03143=1202.868,16.984,-44.194,-179.571,5.622,148.862
C03144=1202.873,16.735,-44.179,-179.573,5.622,148.863
C03145=1202.878,16.486,-44.165,-179.576,5.621,148.863
C03146=1202.883,16.236,-44.150,-179.578,5.621,148.864
C03147=1202.888,15.987,-44.136,-179.581,5.620,148.865
C03148=1202.894,15.737,-44.121,-179.584,5.620,148.866
C03149=1202.898,15.488,-44.106,-179.586,5.619,148.866
C03150=1202.903,15.238,-44.091,-179.589,5.619,148.867
C03151=1202.908,14.988,-44.077,-179.591,5.618,148.867
C03152=1202.913,14.739,-44.062,-179.593,5.618,148.868
C03153=1202.919,14.489,-44.047,-179.596,5.618,148.869
C03154=1202.924,14.239,-44.033,-179.598,5.617,148.869
C03155=1202.928,13.990,-44.018,-179.601,5.616,148.870
C03156=1202.933,13.741,-44.004,-179.603,5.616,148.871
C03157=1202.938,13.491,-43.989,-179.606,5.615,148.871
C03158=1202.943,13.242,-43.974,-179.609,5.615,148.872
C03159=1202.948,12.992,-43.960,-179.611,5.614,148.873
C03160=1202.953,12.742,-43.945,-179.614,5.614,148.873
C03161=1202.959,12.494,-43.931,-179.616,5.613,148.874
C03162=1202.964,12.244,-43.916,-179.619,5.613,148.874
C03163=1202.969,11.994,-43.902,-179.621,5.612,148.875
C03164=1202.974,11.744,-43.888,-179.624,5.612,148.876
C03165=1202.979,11.495,-43.872,-179.626,5.612,148.876
C03166=1202.984,11.245,-43.858,-179.628,5.611,148.877
C03167=1202.989,10.996,-43.844,-179.631,5.610,148.878
C03168=1202.994,10.746,-43.829,-179.634,5.610,148.878
C03169=1202.999,10.496,-43.815,-179.636,5.609,148.879
C03170=1203.004,10.248,-43.801,-179.639,5.609,148.880
C03171=1203.009,9.998,-43.786,-179.642,5.608,148.880
C03172=1203.014,9.748,-43.772,-179.644,5.608,148.881
C03173=1203.019,9.499,-43.758,-179.646,5.607,148.881
C03174=1203.024,9.249,-43.743,-179.649,5.607,148.882
C03175=1203.030,8.999,-43.729,-179.652,5.606,148.883
C03176=1203.034,8.750,-43.714,-179.654,5.606,148.884
C03177=1203.039,8.500,-43.699,-179.656,5.606,148.884
C03178=1203.045,8.251,-43.685,-179.659,5.605,148.885
C03179=1203.050,8.001,-43.671,-179.661,5.604,148.885
C03180=1203.055,7.752,-43.657,-179.664,5.604,148.886
C03181=1203.060,7.502,-43.643,-179.667,5.603,148.887
C03182=1203.065,7.252,-43.628,-179.669,5.603,148.887
C03183=1203.069,7.003,-43.614,-179.672,5.602,148.888
C03184=1203.075,6.754,-43.599,-179.674,5.602,148.889
C03185=1203.080,6.505,-43.585,-179.676,5.602,148.889
C03186=1203.085,6.255,-43.571,-179.679,5.601,148.890
C03187=1203.090,6.005,-43.557,-179.681,5.601,148.891
C03188=1203.095,5.755,-43.542,-179.684,5.600,148.891
C03189=1203.100,5.506,-43.528,-179.687,5.600,148.892
C03190=1203.105,5.257,-43.514,-179.689,5.599,148.892
C03191=1203.110,5.007,-43.500,-179.692,5.599,148.893
C03192=1203.115,4.757,-43.486,-179.694,5.598,148.894
C03193=1203.120,4.508,-43.471,-179.697,5.598,148.895
C03194=1203.125,4.259,-43.457,-179.699,5.598,148.895
C03195=1203.130,4.009,-43.443,-179.702,5.597,148.896
C03196=1203.135,3.759,-43.429,-179.704,5.596,148.896
C03197=1203.140,3.509,-43.415,-179.706,5.596,148.897
C03198=1203.146,3.240,-43.400,-179.709,5.595,148.898
C03199=1203.151,2.972,-43.384,-179.712,5.595,148.898
C03200=1203.157,2.702,-43.369,-179.714,5.594,148.899
C03201=1203.162,2.433,-43.354,-179.717,5.594,148.900
C03202=1203.167,2.183,-43.340,-179.720,5.593,148.900
C03203=1203.172,1.934,-43.326,-179.722,5.593,148.901
C03204=1203.178,1.685,-43.312,-179.725,5.592,148.902
C03205=1203.182,1.435,-43.298,-179.728,5.592,148.903
C03206=1203.187,1.186,-43.284,-179.730,5.592,148.903
C03207=1203.193,0.937,-43.270,-179.732,5.592,148.904
C03208=1203.198,0.687,-43.256,-179.734,5.591,148.904
C03209=1203.202,0.437,-43.241,-179.737,5.590,148.905
C03210=1203.208,0.187,-43.228,-179.740,5.590,148.906
C03211=1203.213,-0.062,-43.214,-179.742,5.589,148.906
C03212=1203.218,-0.312,-43.200,-179.745,5.589,148.907
C03213=1203.222,-0.561,-43.186,-179.747,5.589,148.908
C03214=1203.227,-0.811,-43.172,-179.749,5.588,148.908
C03215=1203.233,-1.060,-43.158,-179.752,5.588,148.909
C03216=1203.238,-1.310,-43.143,-179.755,5.587,148.910
C03217=1203.243,-1.560,-43.130,-179.757,5.587,148.910
C03218=1203.249,-1.809,-43.116,-179.760,5.586,148.911
C03219=1203.253,-2.059,-43.102,-179.763,5.586,148.912
C03220=1203.258,-2.308,-43.088,-179.765,5.586,148.912
C03221=1203.263,-2.557,-43.074,-179.767,5.585,148.913
C03222=1203.269,-2.808,-43.061,-179.769,5.585,148.914
C03223=1203.274,-3.057,-43.046,-179.772,5.584,148.914
C03224=1203.278,-3.306,-43.033,-179.775,5.584,148.915
C03225=1203.283,-3.556,-43.019,-179.777,5.583,148.916
C03226=1203.289,-3.806,-43.005,-179.780,5.583,148.916
C03227=1203.294,-4.055,-42.991,-179.782,5.583,148.917
C03228=1203.299,-4.305,-42.977,-179.784,5.582,148.917
C03229=1203.303,-4.554,-42.963,-179.787,5.582,148.918
C03230=1203.309,-4.804,-42.950,-179.790,5.581,148.919
C03231=1203.314,-5.053,-42.936,-179.792,5.581,148.920
C03232=1203.319,-5.303,-42.921,-179.795,5.580,148.920
C03233=1203.324,-5.553,-42.909,-179.797,5.581,148.921
C03234=1203.329,-5.802,-42.895,-179.799,5.580,148.921
C03235=1203.334,-6.052,-42.880,-179.802,5.579,148.922
C03236=1203.340,-6.302,-42.867,-179.805,5.579,148.923
C03237=1203.344,-6.551,-42.853,-179.807,5.578,148.923
C03238=1203.350,-6.800,-42.840,-179.810,5.578,148.924
C03239=1203.355,-7.050,-42.826,-179.812,5.578,148.925
C03240=1203.359,-7.300,-42.812,-179.815,5.578,148.926
C03241=1203.365,-7.549,-42.798,-179.817,5.577,148.926
C03242=1203.370,-7.799,-42.785,-179.819,5.576,148.927
C03243=1203.375,-8.048,-42.771,-179.822,5.576,148.927
C03244=1203.380,-8.298,-42.758,-179.825,5.575,148.928
C03245=1203.385,-8.548,-42.744,-179.827,5.576,148.929
C03246=1203.390,-8.796,-42.730,-179.829,5.575,148.929
C03247=1203.395,-9.047,-42.717,-179.832,5.575,148.930
C03248=1203.401,-9.296,-42.703,-179.834,5.574,148.931
C03249=1203.405,-9.546,-42.690,-179.837,5.573,148.931
C03250=1203.410,-9.796,-42.676,-179.839,5.574,148.932
C03251=1203.416,-10.045,-42.662,-179.842,5.573,148.933
C03252=1203.420,-10.295,-42.649,-179.844,5.573,148.933
C03253=1203.426,-10.544,-42.635,-179.847,5.572,148.934
C03254=1203.431,-10.794,-42.621,-179.850,5.572,148.935
C03255=1203.436,-11.043,-42.608,-179.851,5.572,148.935
C03256=1203.441,-11.293,-42.594,-179.854,5.571,148.936
C03257=1203.446,-11.542,-42.581,-179.857,5.571,148.937
C03258=1203.451,-11.792,-42.567,-179.859,5.570,148.937
C03259=1203.456,-12.042,-42.553,-179.862,5.570,148.938
C03260=1203.461,-12.291,-42.541,-179.864,5.569,148.939
C03261=1203.467,-12.541,-42.527,-179.867,5.570,148.939
C03262=1203.472,-12.790,-42.514,-179.869,5.569,148.940
C03263=1203.477,-13.040,-42.500,-179.871,5.568,148.941
C03264=1203.482,-13.289,-42.487,-179.874,5.568,148.941
C03265=1203.487,-13.539,-42.473,-179.877,5.567,148.942
C03266=1203.492,-13.788,-42.459,-179.879,5.568,148.943
C03267=1203.497,-14.038,-42.446,-179.881,5.567,148.943
C03268=1203.502,-14.287,-42.433,-179.884,5.567,148.944
C03269=1203.507,-14.537,-42.420,-179.886,5.566,148.944
C03270=1203.513,-14.787,-42.406,-179.889,5.565,148.945
C03271=1203.517,-15.036,-42.393,-179.891,5.566,148.946
C03272=1203.523,-15.286,-42.379,-179.894,5.565,148.947
C03273=1203.527,-15.535,-42.366,-179.896,5.565,148.947
C03274=1203.533,-15.785,-42.353,-179.899,5.564,148.948
C03275=1203.538,-16.035,-42.340,-179.902,5.564,148.949
C03276=1203.543,-16.284,-42.326,-179.903,5.564,148.949
C03277=1203.548,-16.534,-42.313,-179.906,5.563,148.950
C03278=1203.553,-16.784,-42.300,-179.909,5.563,148.950
C03279=1203.558,-17.033,-42.286,-179.911,5.562,148.951
C03280=1203.564,-17.283,-42.273,-179.913,5.563,148.952
C03281=1203.568,-17.533,-42.260,-179.916,5.562,148.953
C03282=1203.574,-17.782,-42.246,-179.919,5.562,148.953
C03283=1203.578,-18.032,-42.233,-179.921,5.561,148.954
C03284=1203.584,-18.281,-42.220,-179.923,5.560,148.954
C03285=1203.589,-18.531,-42.207,-179.925,5.561,148.955
C03286=1203.594,-18.781,-42.193,-179.928,5.560,148.956
C03287=1203.599,-19.030,-42.180,-179.931,5.560,148.957
C03288=1203.604,-19.280,-42.167,-179.933,5.559,148.957
C03289=1203.610,-19.529,-42.154,-179.936,5.559,148.958
C03290=1203.614,-19.779,-42.140,-179.938,5.559,148.959
C03291=1203.620,-20.029,-42.127,-179.940,5.558,148.959
C03292=1203.625,-20.278,-42.115,-179.943,5.558,148.960
C03293=1203.630,-20.528,-42.101,-179.946,5.557,148.960
C03294=1203.635,-20.777,-42.088,-179.948,5.557,148.961
C03295=1203.639,-21.027,-42.075,-179.950,5.557,148.962
C03296=1203.645,-21.277,-42.061,-179.953,5.557,148.963
C03297=1203.650,-21.526,-42.049,-179.956,5.556,148.963
C03298=1203.656,-21.776,-42.035,-179.957,5.556,148.964
C03299=1203.660,-22.025,-42.022,-179.960,5.556,148.964
C03300=1203.665,-22.275,-42.009,-179.963,5.555,148.965
C03301=1203.671,-22.525,-41.996,-179.965,5.555,148.966
C03302=1203.676,-22.794,-41.982,-179.968,5.554,148.966
C03303=1203.682,-23.064,-41.968,-179.971,5.554,148.967
C03304=1203.687,-23.333,-41.954,-179.973,5.554,148.968
C03305=1203.693,-23.603,-41.940,-179.975,5.553,148.969
C03306=1203.698,-23.852,-41.927,-179.978,5.553,148.969
C03307=1203.703,-24.102,-41.913,-179.981,5.553,148.970
C03308=1203.708,-24.352,-41.901,-179.983,5.552,148.971
C03309=1203.713,-24.601,-41.888,-179.985,5.552,148.971
C03310=1203.719,-24.851,-41.875,-179.988,5.552,148.972
C03311=1203.723,-25.100,-41.861,-179.991,5.551,148.973
C03312=1203.728,-25.349,-41.849,-179.993,5.551,148.973
C03313=1203.733,-25.599,-41.836,-179.995,5.551,148.974
C03314=1203.739,-25.849,-41.823,-179.998,5.550,148.975
C03315=1203.744,-26.098,-41.810,180.000,5.550,148.975
C03316=1203.749,-26.348,-41.797,179.997,5.550,148.976
C03317=1203.754,-26.598,-41.784,179.995,5.550,148.977
C03318=1203.760,-26.847,-41.771,179.992,5.549,148.977
C03319=1203.764,-27.097,-41.758,179.990,5.549,148.978
C03320=1203.769,-27.347,-41.746,179.987,5.548,148.979
C03321=1203.775,-27.596,-41.732,179.985,5.548,148.979
C03322=1203.780,-27.846,-41.719,179.983,5.548,148.980
C03323=1203.785,-28.096,-41.707,179.980,5.547,148.981
C03324=1203.790,-28.345,-41.694,179.977,5.547,148.981
C03325=1203.795,-28.595,-41.681,179.975,5.547,148.982
C03326=1203.800,-28.845,-41.668,179.973,5.547,148.983
C03327=1203.805,-29.094,-41.656,179.970,5.546,148.983
C03328=1203.810,-29.343,-41.643,179.968,5.546,148.984
C03329=1203.815,-29.593,-41.630,179.966,5.546,148.985
C03330=1203.821,-29.843,-41.617,179.963,5.545,148.985
C03331=1203.826,-30.092,-41.604,179.960,5.545,148.986
C03332=1203.831,-30.343,-41.592,179.958,5.544,148.987
C03333=1203.836,-30.592,-41.579,179.956,5.545,148.987
C03334=1203.841,-30.841,-41.567,179.954,5.544,148.988
C03335=1203.847,-31.091,-41.553,179.951,5.543,148.989
C03336=1203.851,-31.341,-41.541,179.949,5.544,148.989
C03337=1203.857,-31.590,-41.528,179.946,5.543,148.990
C03338=1203.862,-31.840,-41.515,179.943,5.543,148.991
C03339=1203.867,-32.089,-41.503,179.941,5.542,148.991
C03340=1203.871,-32.339,-41.490,179.939,5.543,148.992
C03341=1203.877,-32.589,-41.477,179.936,5.542,148.993
C03342=1203.883,-32.839,-41.465,179.934,5.541,148.993
C03343=1203.888,-33.088,-41.452,179.931,5.541,148.994
C03344=1203.892,-33.338,-41.439,179.929,5.541,148.995
C03345=1203.897,-33.587,-41.427,179.926,5.541,148.995
C03346=1203.902,-33.837,-41.414,179.924,5.540,148.996
C03347=1203.908,-34.086,-41.402,179.922,5.541,148.997
C03348=1203.912,-34.337,-41.389,179.919,5.540,148.997
C03349=1203.918,-34.586,-41.376,179.917,5.539,148.998
C03350=1203.923,-34.835,-41.363,179.914,5.539,148.999
C03351=1203.929,-35.085,-41.351,179.912,5.539,148.999
C03352=1203.934,-35.335,-41.339,179.909,5.539,149.000
C03353=1203.938,-35.585,-41.326,179.907,5.538,149.001
C03354=1203.944,-35.834,-41.313,179.905,5.539,149.001
C03355=1203.949,-36.083,-41.301,179.902,5.538,149.002
C03356=1203.954,-36.333,-41.289,179.900,5.537,149.003
C03357=1203.959,-36.583,-41.276,179.897,5.537,149.003
C03358=1203.964,-36.833,-41.263,179.895,5.537,149.004
C03359=1203.969,-37.083,-41.251,179.893,5.537,149.005
C03360=1203.974,-37.332,-41.239,179.890,5.536,149.005
C03361=1203.979,-37.581,-41.226,179.888,5.537,149.006
C03362=1203.985,-37.831,-41.213,179.885,5.536,149.007
C03363=1203.991,-38.081,-41.201,179.882,5.536,149.007
C03364=1203.995,-38.331,-41.188,179.880,5.535,149.008
C03365=1204.000,-38.580,-41.175,179.878,5.535,149.009
C03366=1204.006,-38.830,-41.164,179.876,5.535,149.009
C03367=1204.011,-39.079,-41.151,179.873,5.534,149.010
C03368=1204.016,-39.329,-41.138,179.871,5.535,149.011
C03369=1204.022,-39.579,-41.126,179.868,5.534,149.011
C03370=1204.027,-39.828,-41.114,179.865,5.534,149.012
C03371=1204.031,-40.078,-41.101,179.864,5.534,149.013
C03372=1204.037,-40.328,-41.089,179.861,5.533,149.013
C03373=1204.042,-40.577,-41.076,179.859,5.533,149.014
C03374=1204.047,-40.827,-41.065,179.856,5.532,149.015
C03375=1204.052,-41.076,-41.053,179.854,5.533,149.015
C03376=1204.057,-41.325,-41.040,179.851,5.532,149.016
C03377=1204.062,-41.575,-41.028,179.848,5.532,149.017
C03378=1204.067,-41.825,-41.015,179.847,5.532,149.017
C03379=1204.072,-42.075,-41.003,179.844,5.531,149.018
C03380=1204.077,-42.325,-40.991,179.842,5.531,149.019
C03381=1204.083,-42.575,-40.979,179.839,5.531,149.019
C03382=1204.088,-42.824,-40.966,179.837,5.531,149.020
C03383=1204.093,-43.074,-40.954,179.834,5.530,149.021
C03384=1204.098,-43.323,-40.942,179.832,5.530,149.021
C03385=1204.103,-43.573,-40.929,179.830,5.530,149.022
C03386=1204.109,-43.822,-40.917,179.827,5.529,149.023
C03387=1204.114,-44.072,-40.905,179.825,5.530,149.023
C03388=1204.119,-44.322,-40.893,179.822,5.529,149.024
C03389=1204.124,-44.571,-40.881,179.820,5.529,149.025
C03390=1204.129,-44.821,-40.869,179.817,5.528,149.025
C03391=1204.134,-45.071,-40.856,179.815,5.528,149.026
C03392=1204.139,-45.321,-40.844,179.813,5.528,149.027
C03393=1204.145,-45.571,-40.832,179.810,5.527,149.027
C03394=1204.150,-45.820,-40.819,179.808,5.528,149.028
C03395=1204.155,-46.070,-40.808,179.805,5.527,149.029
C03396=1204.160,-46.319,-40.795,179.803,5.527,149.029
C03397=1204.165,-46.569,-40.784,179.801,5.527,149.030
C03398=1204.170,-46.818,-40.771,179.798,5.527,149.031
C03399=1204.176,-47.068,-40.759,179.796,5.526,149.031
C03400=1204.181,-47.317,-40.747,179.794,5.526,149.032
C03401=1204.186,-47.567,-40.735,179.791,5.526,149.033
C03402=1204.191,-47.817,-40.723,179.788,5.525,149.033
C03403=1204.196,-48.066,-40.711,179.786,5.525,149.034
C03404=1204.201,-48.316,-40.699,179.784,5.525,149.035
C03405=1204.207,-48.566,-40.687,179.781,5.525,149.036
C03406=1204.212,-48.836,-40.673,179.779,5.525,149.036
C03407=1204.218,-49.105,-40.661,179.776,5.524,149.037
C03408=1204.223,-49.376,-40.648,179.774,5.524,149.038
C03409=1204.229,-49.646,-40.634,179.771,5.524,149.038
C03410=1204.234,-49.896,-40.623,179.769,5.524,149.039
C03411=1204.239,-50.145,-40.610,179.766,5.523,149.040
C03412=1204.244,-50.395,-40.598,179.764,5.523,149.040
C03413=1204.250,-50.645,-40.587,179.762,5.523,149.041
C03414=1204.254,-50.894,-40.575,179.759,5.522,149.042
C03415=1204.259,-51.144,-40.563,179.757,5.522,149.042
C03416=1204.265,-51.394,-40.551,179.755,5.522,149.043
C03417=1204.270,-51.644,-40.539,179.752,5.522,149.044
C03418=1204.275,-51.893,-40.527,179.749,5.521,149.044
C03419=1204.281,-52.142,-40.515,179.747,5.522,149.045
C03420=1204.286,-52.392,-40.503,179.745,5.521,149.046
C03421=1204.291,-52.642,-40.491,179.742,5.521,149.046
C03422=1204.296,-52.891,-40.480,179.740,5.521,149.047
C03423=1204.301,-53.141,-40.468,179.738,5.520,149.048
C03424=1204.307,-53.391,-40.456,179.735,5.520,149.048
C03425=1204.311,-53.640,-40.444,179.733,5.520,149.049
C03426=1204.317,-53.890,-40.432,179.731,5.520,149.050
C03427=1204.322,-54.140,-40.420,179.728,5.519,149.050
C03428=1204.327,-54.390,-40.409,179.726,5.519,149.051
C03429=1204.332,-54.640,-40.397,179.723,5.519,149.052
C03430=1204.337,-54.889,-40.384,179.721,5.519,149.052
C03431=1204.342,-55.138,-40.373,179.718,5.519,149.053
C03432=1204.347,-55.388,-40.361,179.716,5.518,149.054
C03433=1204.353,-55.638,-40.349,179.714,5.518,149.054
C03434=1204.358,-55.888,-40.338,179.712,5.518,149.055
C03435=1204.363,-56.138,-40.326,179.709,5.517,149.056
C03436=1204.368,-56.387,-40.313,179.707,5.518,149.056
C03437=1204.373,-56.636,-40.302,179.704,5.517,149.057
C03438=1204.379,-56.886,-40.291,179.701,5.517,149.058
C03439=1204.384,-57.136,-40.279,179.699,5.517,149.059
C03440=1204.389,-57.386,-40.267,179.697,5.516,149.059
C03441=1204.394,-57.636,-40.256,179.694,5.516,149.060
C03442=1204.399,-57.885,-40.244,179.692,5.516,149.060
C03443=1204.405,-58.135,-40.232,179.690,5.516,149.061
C03444=1204.410,-58.384,-40.220,179.687,5.515,149.062
C03445=1204.414,-58.634,-40.208,179.685,5.516,149.063
C03446=1204.420,-58.883,-40.197,179.683,5.515,149.063
C03447=1204.425,-59.133,-40.186,179.681,5.515,149.064
C03448=1204.431,-59.383,-40.174,179.678,5.515,149.064
C03449=1204.435,-59.633,-40.162,179.675,5.514,149.065
C03450=1204.441,-59.882,-40.151,179.673,5.515,149.066
C03451=1204.446,-60.132,-40.139,179.671,5.514,149.067
C03452=1204.451,-60.382,-40.127,179.668,5.514,149.067
C03453=1204.456,-60.632,-40.116,179.666,5.514,149.068
C03454=1204.461,-60.881,-40.105,179.664,5.513,149.068
C03455=1204.467,-61.131,-40.093,179.662,5.514,149.069
C03456=1204.472,-61.380,-40.081,179.659,5.513,149.070
C03457=1204.477,-61.630,-40.070,179.656,5.513,149.071
C03458=1204.482,-61.880,-40.058,179.654,5.513,149.071
C03459=1204.487,-62.130,-40.046,179.652,5.512,149.072
C03460=1204.492,-62.379,-40.035,179.649,5.512,149.072
C03461=1204.498,-62.629,-40.024,179.647,5.512,149.073
C03462=1204.503,-62.878,-40.012,179.645,5.512,149.074
C03463=1204.508,-63.128,-40.000,179.643,5.512,149.075
C03464=1204.513,-63.378,-39.989,179.640,5.512,149.075
C03465=1204.519,-63.627,-39.978,179.638,5.511,149.076
C03466=1204.523,-63.877,-39.966,179.636,5.511,149.076
C03467=1204.529,-64.127,-39.954,179.633,5.511,149.077
C03468=1204.534,-64.376,-39.943,179.630,5.510,149.078
C03469=1204.539,-64.626,-39.931,179.628,5.511,149.079
C03470=1204.545,-64.876,-39.921,179.626,5.510,149.079
C03471=1204.550,-65.126,-39.909,179.624,5.510,149.080
C03472=1204.555,-65.375,-39.898,179.621,5.510,149.080
C03473=1204.560,-65.625,-39.886,179.619,5.510,149.081
C03474=1204.565,-65.875,-39.875,179.616,5.510,149.082
C03475=1204.571,-66.124,-39.863,179.614,5.509,149.083
C03476=1204.576,-66.374,-39.852,179.612,5.510,149.083
C03477=1204.580,-66.623,-39.841,179.610,5.509,149.084
C03478=1204.586,-66.874,-39.829,179.607,5.509,149.084
C03479=1204.591,-67.123,-39.818,179.605,5.509,149.085
C03480=1204.597,-67.373,-39.807,179.602,5.508,149.086
C03481=1204.601,-67.623,-39.795,179.600,5.509,149.087
C03482=1204.607,-67.872,-39.783,179.597,5.508,149.087
C03483=1204.612,-68.121,-39.772,179.595,5.508,149.088
C03484=1204.617,-68.372,-39.762,179.593,5.508,149.088
C03485=1204.623,-68.622,-39.750,179.590,5.507,149.089
C03486=1204.627,-68.871,-39.739,179.588,5.508,149.090
C03487=1204.633,-69.120,-39.727,179.586,5.507,149.091
C03488=1204.638,-69.371,-39.717,179.583,5.507,149.091
C03489=1204.643,-69.620,-39.705,179.581,5.507,149.092
C03490=1204.648,-69.870,-39.693,179.579,5.506,149.092
C03491=1204.654,-70.119,-39.683,179.577,5.507,149.093
C03492=1204.659,-70.369,-39.672,179.574,5.506,149.094
C03493=1204.664,-70.619,-39.660,179.571,5.506,149.095
C03494=1204.669,-70.868,-39.649,179.570,5.506,149.095
C03495=1204.674,-71.118,-39.638,179.567,5.506,149.096
C03496=1204.680,-71.368,-39.627,179.565,5.506,149.096
C03497=1204.684,-71.618,-39.615,179.562,5.505,149.097
C03498=1204.690,-71.867,-39.604,179.560,5.505,149.098
C03499=1204.695,-72.117,-39.593,179.558,5.505,149.099
C03500=1204.700,-72.367,-39.582,179.555,5.505,149.099
C03501=1204.705,-72.616,-39.571,179.553,5.505,149.100
C03502=1204.711,-72.866,-39.559,179.551,5.504,149.101
C03503=1204.716,-73.116,-39.549,179.548,5.504,149.101
C03504=1204.721,-73.365,-39.538,179.546,5.504,149.102
C03505=1204.727,-73.615,-39.526,179.543,5.504,149.103
C03506=1204.732,-73.865,-39.515,179.542,5.504,149.103
C03507=1204.737,-74.114,-39.504,179.539,5.504,149.104
C03508=1204.742,-74.365,-39.494,179.537,5.504,149.105
C03509=1204.747,-74.615,-39.482,179.534,5.503,149.105
C03510=1204.754,-74.885,-39.470,179.531,5.503,149.106
C03511=1204.758,-75.155,-39.458,179.529,5.503,149.107
C03512=1204.765,-75.426,-39.446,179.527,5.503,149.107
C03513=1204.770,-75.697,-39.434,179.524,5.503,149.108
C03514=1204.775,-75.946,-39.423,179.522,5.503,149.109
C03515=1204.781,-76.196,-39.413,179.519,5.502,149.109
C03516=1204.786,-76.446,-39.401,179.517,5.502,149.110
C03517=1204.791,-76.696,-39.390,179.515,5.502,149.111
C03518=1204.796,-76.945,-39.379,179.512,5.502,149.111
C03519=1204.801,-77.195,-39.369,179.510,5.502,149.112
C03520=1204.807,-77.444,-39.358,179.508,5.502,149.113
C03521=1204.812,-77.694,-39.346,179.505,5.501,149.113
C03522=1204.817,-77.944,-39.335,179.503,5.501,149.114
C03523=1204.822,-78.193,-39.324,179.501,5.501,149.115
C03524=1204.827,-78.444,-39.314,179.499,5.501,149.115
C03525=1204.832,-78.693,-39.303,179.496,5.501,149.116
C03526=1204.838,-78.943,-39.292,179.494,5.501,149.117
C03527=1204.843,-79.193,-39.280,179.492,5.500,149.117
C03528=1204.849,-79.442,-39.270,179.489,5.500,149.118
C03529=1204.853,-79.692,-39.259,179.487,5.500,149.119
C03530=1204.859,-79.941,-39.249,179.484,5.500,149.119
C03531=1204.864,-80.191,-39.237,179.482,5.500,149.120
C03532=1204.869,-80.442,-39.226,179.480,5.499,149.121
C03533=1204.875,-80.691,-39.216,179.478,5.500,149.121
C03534=1204.880,-80.941,-39.205,179.475,5.499,149.122
C03535=1204.885,-81.190,-39.195,179.473,5.499,149.123
C03536=1204.890,-81.440,-39.183,179.470,5.499,149.123
C03537=1204.895,-81.690,-39.173,179.468,5.498,149.124
C03538=1204.900,-81.939,-39.162,179.466,5.499,149.125
C03539=1204.906,-82.190,-39.151,179.463,5.498,149.125
C03540=1204.912,-82.439,-39.140,179.461,5.499,149.126
C03541=1204.916,-82.689,-39.129,179.459,5.498,149.127
C03542=1204.922,-82.938,-39.119,179.457,5.498,149.127
C03543=1204.927,-83.188,-39.108,179.454,5.498,149.128
C03544=1204.932,-83.437,-39.097,179.452,5.497,149.129
C03545=1204.937,-83.688,-39.087,179.450,5.498,149.129
C03546=1204.942,-83.937,-39.076,179.447,5.497,149.130
C03547=1204.947,-84.187,-39.065,179.445,5.497,149.131
C03548=1204.952,-84.436,-39.054,179.443,5.497,149.131
C03549=1204.958,-84.686,-39.044,179.441,5.497,149.132
C03550=1204.963,-84.936,-39.033,179.438,5.497,149.133
C03551=1204.969,-85.186,-39.022,179.436,5.497,149.133
C03552=1204.974,-85.436,-39.011,179.434,5.496,149.134
C03553=1204.979,-85.685,-39.001,179.431,5.496,149.135
C03554=1204.984,-85.935,-38.990,179.429,5.496,149.135
C03555=1204.990,-86.184,-38.979,179.426,5.496,149.136
C03556=1204.995,-86.435,-38.969,179.425,5.496,149.137
C03557=1205.000,-86.684,-38.959,179.422,5.495,149.137
C03558=1205.005,-86.934,-38.947,179.420,5.496,149.138
C03559=1205.011,-87.183,-38.937,179.417,5.495,149.139
C03560=1205.016,-87.434,-38.927,179.415,5.496,149.139
C03561=1205.021,-87.683,-38.916,179.413,5.495,149.140
C03562=1205.026,-87.933,-38.905,179.411,5.495,149.141
C03563=1205.031,-88.182,-38.895,179.408,5.495,149.141
C03564=1205.036,-88.433,-38.884,179.406,5.494,149.142
C03565=1205.042,-88.682,-38.873,179.403,5.495,149.143
C03566=1205.047,-88.931,-38.863,179.401,5.494,149.143
C03567=1205.052,-89.181,-38.853,179.399,5.494,149.144
C03568=1205.058,-89.431,-38.842,179.397,5.494,149.145
C03569=1205.063,-89.681,-38.832,179.394,5.494,149.145
C03570=1205.068,-89.930,-38.821,179.392,5.493,149.146
C03571=1205.073,-90.180,-38.810,179.390,5.494,149.146
C03572=1205.079,-90.430,-38.800,179.387,5.493,149.147
C03573=1205.083,-90.680,-38.790,179.385,5.494,149.148
C03574=1205.089,-90.929,-38.780,179.383,5.493,149.149
C03575=1205.093,-91.179,-38.769,179.381,5.493,149.149
C03576=1205.099,-91.428,-38.758,179.378,5.493,149.150
C03577=1205.105,-91.678,-38.748,179.376,5.493,149.151
C03578=1205.110,-91.928,-38.738,179.374,5.493,149.151
C03579=1205.115,-92.178,-38.727,179.372,5.492,149.152
C03580=1205.120,-92.428,-38.717,179.369,5.492,149.152
C03581=1205.126,-92.678,-38.707,179.367,5.492,149.153
C03582=1205.130,-92.927,-38.695,179.365,5.492,149.154
C03583=1205.136,-93.177,-38.685,179.362,5.492,149.154
C03584=1205.142,-93.426,-38.675,179.360,5.492,149.155
C03585=1205.147,-93.677,-38.664,179.358,5.492,149.156
C03586=1205.151,-93.926,-38.655,179.356,5.492,149.156
C03587=1205.156,-94.176,-38.644,179.353,5.492,149.157
C03588=1205.162,-94.426,-38.634,179.351,5.492,149.158
C03589=1205.168,-94.675,-38.624,179.349,5.491,149.158
C03590=1205.173,-94.925,-38.613,179.346,5.491,149.159
C03591=1205.178,-95.175,-38.603,179.344,5.491,149.160
C03592=1205.184,-95.424,-38.593,179.342,5.490,149.160
C03593=1205.188,-95.674,-38.583,179.340,5.491,149.161
C03594=1205.194,-95.924,-38.573,179.337,5.490,149.162
C03595=1205.199,-96.174,-38.562,179.335,5.491,149.162
C03596=1205.204,-96.423,-38.551,179.333,5.490,149.163
C03597=1205.210,-96.673,-38.541,179.331,5.490,149.164
C03598=1205.215,-96.923,-38.530,179.328,5.490,149.164
C03599=1205.220,-97.172,-38.520,179.326,5.490,149.165
C03600=1205.225,-97.422,-38.511,179.324,5.489,149.166
C03601=1205.230,-97.672,-38.500,179.322,5.490,149.166
C03602=1205.236,-97.921,-38.490,179.319,5.489,149.167
C03603=1205.242,-98.172,-38.480,179.317,5.490,149.168
C03604=1205.247,-98.422,-38.470,179.315,5.489,149.168
C03605=1205.251,-98.671,-38.460,179.313,5.489,149.169
C03606=1205.257,-98.921,-38.450,179.310,5.489,149.170
C03607=1205.262,-99.171,-38.439,179.308,5.489,149.170
C03608=1205.268,-99.420,-38.429,179.306,5.488,149.171
C03609=1205.273,-99.670,-38.419,179.304,5.489,149.171
C03610=1205.277,-99.920,-38.409,179.301,5.488,149.172
C03611=1205.283,-100.169,-38.399,179.299,5.489,149.173
C03612=1205.289,-100.419,-38.388,179.297,5.488,149.173
C03613=1205.294,-100.669,-38.378,179.294,5.488,149.174
C03614=1205.299,-100.940,-38.367,179.292,5.488,149.175
C03615=1205.305,-101.211,-38.356,179.289,5.488,149.176
C03616=1205.311,-101.483,-38.346,179.287,5.488,149.176
C03617=1205.316,-101.755,-38.335,179.284,5.488,149.177
C03618=1205.322,-102.004,-38.324,179.282,5.487,149.178
C03619=1205.327,-102.254,-38.314,179.280,5.488,149.178
C03620=1205.332,-102.503,-38.305,179.277,5.487,149.179
C03621=1205.337,-102.753,-38.294,179.275,5.487,149.180
C03622=1205.343,-103.003,-38.284,179.273,5.487,149.180
C03623=1205.348,-103.253,-38.275,179.271,5.487,149.181
C03624=1205.353,-103.503,-38.264,179.268,5.486,149.181
C03625=1205.358,-103.752,-38.254,179.266,5.487,149.182
C03626=1205.363,-104.002,-38.244,179.264,5.486,149.183
C03627=1205.369,-104.251,-38.234,179.262,5.486,149.183
C03628=1205.374,-104.501,-38.224,179.259,5.486,149.184
C03629=1205.379,-104.751,-38.215,179.257,5.486,149.185
C03630=1205.385,-105.001,-38.205,179.255,5.486,149.186
C03631=1205.390,-105.250,-38.194,179.253,5.486,149.186
C03632=1205.395,-105.500,-38.184,179.250,5.485,149.187
C03633=1205.400,-105.750,-38.175,179.248,5.486,149.187
C03634=1205.406,-106.000,-38.165,179.245,5.485,149.188
C03635=1205.411,-106.249,-38.155,179.244,5.485,149.189
C03636=1205.416,-106.499,-38.145,179.241,5.485,149.189
C03637=1205.421,-106.749,-38.134,179.239,5.485,149.190
C03638=1205.427,-106.999,-38.125,179.237,5.485,149.191
C03639=1205.432,-107.248,-38.115,179.235,5.485,149.191
C03640=1205.437,-107.499,-38.105,179.232,5.485,149.192
C03641=1205.442,-107.749,-38.096,179.230,5.485,149.193
C03642=1205.448,-107.998,-38.086,179.228,5.484,149.193
C03643=1205.453,-108.247,-38.076,179.226,5.484,149.194
C03644=1205.458,-108.497,-38.066,179.223,5.484,149.195
C03645=1205.464,-108.748,-38.056,179.221,5.484,149.195
C03646=1205.469,-108.997,-38.046,179.219,5.484,149.196
